LIN {X 0,Y 259.453,Z 689.028,A -85,B 0,C 180,E1 -16715.299,E2 -16715.299} C_VEL
LIN {X 0,Y 272.346,Z 664.838,A -85,B 0,C 180,E1 -16716.608,E2 -16716.608} C_VEL
LIN {X 0,Y 275.458,Z 659.109,A -85,B 0,C 180,E1 -16716.892,E2 -16716.892} C_VEL
LIN {X 0,Y 274.877,Z 634.76,A -85,B 0,C 180,E1 -16720.781,E2 -16720.781} C_VEL
LIN {X 0,Y 277.063,Z 609.313,A -85,B 0,C 180,E1 -16724.48,E2 -16724.48} C_VEL
LIN {X 0,Y 280.601,Z 587.916,A -85,B 0,C 180,E1 -16727.342,E2 -16727.342} C_VEL
LIN {X 0,Y 272.817,Z 572.023,A -85,B 0,C 180,E1 -16732.207,E2 -16732.207} C_VEL
LIN {X 0,Y 265.765,Z 558.11,A -85,B 0,C 180,E1 -16736.981,E2 -16736.981} C_VEL
LIN {X 0,Y 259.589,Z 546.11,A -85,B 0,C 180,E1 -16741.546,E2 -16741.546} C_VEL
LIN {X 0,Y 252.838,Z 533.27,A -85,B 0,C 180,E1 -16746.983,E2 -16746.983} C_VEL
LIN {X 0,Y 246.707,Z 521.951,A -85,B 0,C 180,E1 -16752.404,E2 -16752.404} C_VEL
LIN {X 0,Y 244.594,Z 517.879,A -85,B 0,C 180,E1 -16754.553,E2 -16754.553} C_VEL
LIN {X 0,Y 250.997,Z 514.698,A -85,B 0,C 180,E1 -16759.308,E2 -16759.308} C_VEL
LIN {X 0,Y 255.933,Z 513.422,A -85,B 0,C 180,E1 -16762.33,E2 -16762.33} C_VEL
LIN {X 0,Y 259.283,Z 523.373,A -85,B 0,C 180,E1 -16766.08,E2 -16766.08} C_VEL
LIN {X 0,Y 261.952,Z 531.547,A -85,B 0,C 180,E1 -16768.56,E2 -16768.56} C_VEL
LIN {X 0,Y 265.003,Z 538.596,A -85,B 0,C 180,E1 -16770.186,E2 -16770.186} C_VEL
LIN {X 0,Y 250.876,Z 717.726,A -85,B 0,C 180,E1 -16774.443,E2 -16774.443} C_VEL
LIN {X 0,Y 249.12,Z 743.516,A -85,B 0,C 180,E1 -16775.324,E2 -16775.324} C_VEL
LIN {X 0,Y 246.678,Z 762.04,A -85,B 0,C 180,E1 -16776.293,E2 -16776.293} C_VEL
LIN {X 0,Y 243.283,Z 779.25,A -85,B 0,C 180,E1 -16777.515,E2 -16777.515} C_VEL
LIN {X 0,Y 238.857,Z 796.037,A -85,B 0,C 180,E1 -16779.059,E2 -16779.059} C_VEL
LIN {X 0,Y 233.621,Z 812.02,A -85,B 0,C 180,E1 -16780.941,E2 -16780.941} C_VEL
LIN {X 0,Y 227.692,Z 827.174,A -85,B 0,C 180,E1 -16783.202,E2 -16783.202} C_VEL
LIN {X 0,Y 221.171,Z 841.428,A -85,B 0,C 180,E1 -16785.878,E2 -16785.878} C_VEL
LIN {X 0,Y 214.515,Z 854.248,A -85,B 0,C 180,E1 -16788.914,E2 -16788.914} C_VEL
LIN {X 0,Y 207.446,Z 866.472,A -85,B 0,C 180,E1 -16792.606,E2 -16792.606} C_VEL
LIN {X 0,Y 200.467,Z 877.488,A -85,B 0,C 180,E1 -16796.923,E2 -16796.923} C_VEL
LIN {X 0,Y 194.271,Z 886.647,A -85,B 0,C 180,E1 -16801.655,E2 -16801.655} C_VEL
LIN {X 0,Y 189.179,Z 893.877,A -85,B 0,C 180,E1 -16806.648,E2 -16806.648} C_VEL
LIN {X 0,Y 185.088,Z 899.588,A -85,B 0,C 180,E1 -16812.067,E2 -16812.067} C_VEL
LIN {X 0,Y 182.155,Z 903.783,A -85,B 0,C 180,E1 -16817.962,E2 -16817.962} C_VEL
LIN {X 0,Y 180.522,Z 906.241,A -85,B 0,C 180,E1 -16823.96,E2 -16823.96} C_VEL
LIN {X 0,Y 180.001,Z 907.066,A -85,B 0,C 180,E1 -16830.001,E2 -16830.001} C_VEL
LIN {X 0,Y 180.511,Z 906.288,A -85,B 0,C 180,E1 -16836.042,E2 -16836.042} C_VEL
LIN {X 0,Y 182.13,Z 903.873,A -85,B 0,C 180,E1 -16842.042,E2 -16842.042} C_VEL
LIN {X 0,Y 185.046,Z 899.716,A -85,B 0,C 180,E1 -16847.939,E2 -16847.939} C_VEL
LIN {X 0,Y 189.122,Z 894.048,A -85,B 0,C 180,E1 -16853.361,E2 -16853.361} C_VEL
LIN {X 0,Y 194.121,Z 886.989,A -85,B 0,C 180,E1 -16858.286,E2 -16858.286} C_VEL
LIN {X 0,Y 200.221,Z 878.015,A -85,B 0,C 180,E1 -16862.979,E2 -16862.979} C_VEL
LIN {X 0,Y 206.911,Z 867.529,A -85,B 0,C 180,E1 -16867.161,E2 -16867.161} C_VEL
LIN {X 0,Y 213.926,Z 855.521,A -85,B 0,C 180,E1 -16870.871,E2 -16870.871} C_VEL
LIN {X 0,Y 221.067,Z 841.893,A -85,B 0,C 180,E1 -16874.15,E2 -16874.15} C_VEL
LIN {X 0,Y 227.589,Z 827.727,A -85,B 0,C 180,E1 -16876.827,E2 -16876.827} C_VEL
LIN {X 0,Y 233.404,Z 813.001,A -85,B 0,C 180,E1 -16879.047,E2 -16879.047} C_VEL
LIN {X 0,Y 236.682,Z 803.474,A -85,B 0,C 180,E1 -16880.252,E2 -16880.252} C_VEL
LIN {X 0,Y 233.357,Z 806.151,A -85,B 0,C 180,E1 -16880.786,E2 -16880.786} C_VEL
LIN {X 0,Y 228.962,Z 810.608,A -85,B 0,C 180,E1 -16881.294,E2 -16881.294} C_VEL
LIN {X 0,Y 219.978,Z 819.575,A -85,B 0,C 180,E1 -16882.275,E2 -16882.275} C_VEL
LIN {X 0,Y 210.065,Z 829.053,A -85,B 0,C 180,E1 -16883.348,E2 -16883.348} C_VEL
LIN {X 0,Y 204.628,Z 833.297,A -85,B 0,C 180,E1 -16884.258,E2 -16884.258} C_VEL
LIN {X 0,Y 199.638,Z 836.307,A -85,B 0,C 180,E1 -16885.531,E2 -16885.531} C_VEL
LIN {X 0,Y 197.045,Z 837.699,A -85,B 0,C 180,E1 -16886.325,E2 -16886.325} C_VEL
LIN {X 0,Y 192.369,Z 840.67,A -85,B 0,C 180,E1 -16887.631,E2 -16887.631} C_VEL
LIN {X 0,Y 189.154,Z 842.143,A -85,B 0,C 180,E1 -16888.908,E2 -16888.908} C_VEL
LIN {X 0,Y 185.107,Z 844.669,A -85,B 0,C 180,E1 -16890.201,E2 -16890.201} C_VEL
LIN {X 0,Y 182.785,Z 845.372,A -85,B 0,C 180,E1 -16891.536,E2 -16891.536} C_VEL
LIN {X 0,Y 179.182,Z 860.953,A -85,B 0,C 180,E1 -16895.61,E2 -16895.61} C_VEL
LIN {X 0,Y 176.145,Z 874.608,A -85,B 0,C 180,E1 -16900.087,E2 -16900.087} C_VEL
LIN {X 0,Y 173.819,Z 886.537,A -85,B 0,C 180,E1 -16904.997,E2 -16904.997} C_VEL
LIN {X 0,Y 172.437,Z 896.396,A -85,B 0,C 180,E1 -16909.981,E2 -16909.981} C_VEL
LIN {X 0,Y 171.971,Z 905.792,A -85,B 0,C 180,E1 -16915.998,E2 -16915.998} C_VEL
LIN {X 0,Y 172.771,Z 912.99,A -85,B 0,C 180,E1 -16921.989,E2 -16921.989} C_VEL
LIN {X 0,Y 174.945,Z 918.343,A -85,B 0,C 180,E1 -16927.883,E2 -16927.883} C_VEL
LIN {X 0,Y 178.913,Z 922.183,A -85,B 0,C 180,E1 -16933.904,E2 -16933.904} C_VEL
LIN {X 0,Y 185.401,Z 924.385,A -85,B 0,C 180,E1 -16940.19,E2 -16940.19} C_VEL
LIN {X 0,Y 194.533,Z 924.651,A -85,B 0,C 180,E1 -16946.232,E2 -16946.232} C_VEL
LIN {X 0,Y 205.919,Z 923.034,A -85,B 0,C 180,E1 -16951.627,E2 -16951.627} C_VEL
LIN {X 0,Y 216.667,Z 920.548,A -85,B 0,C 180,E1 -16955.552,E2 -16955.552} C_VEL
LIN {X 0,Y 197.139,Z 933.33,A -85,B 0,C 180,E1 -16962.813,E2 -16962.813} C_VEL
LIN {X 0,Y 182.526,Z 944.843,A -85,B 0,C 180,E1 -16971.755,E2 -16971.755} C_VEL
LIN {X 0,Y 174.003,Z 953.57,A -85,B 0,C 180,E1 -16981.138,E2 -16981.138} C_VEL
LIN {X 0,Y 170.524,Z 959.101,A -85,B 0,C 180,E1 -16989.401,E2 -16989.401} C_VEL
LIN {X 0,Y 169.853,Z 962.452,A -85,B 0,C 180,E1 -16997.073,E2 -16997.073} C_VEL
LIN {X 0,Y 170.554,Z 963.775,A -85,B 0,C 180,E1 -17003.266,E2 -17003.266} C_VEL
LIN {X 0,Y 171.282,Z 963.757,A -85,B 0,C 180,E1 -17007.992,E2 -17007.992} C_VEL
LIN {X 0,Y 171.409,Z 963.117,A -85,B 0,C 180,E1 -17012.005,E2 -17012.005} C_VEL
LIN {X 0,Y 170.864,Z 961.986,A -85,B 0,C 180,E1 -17016.72,E2 -17016.72} C_VEL
LIN {X 0,Y 170.36,Z 959.287,A -85,B 0,C 180,E1 -17022.197,E2 -17022.197} C_VEL
LIN {X 0,Y 170.676,Z 954.511,A -85,B 0,C 180,E1 -17028.441,E2 -17028.441} C_VEL
LIN {X 0,Y 172.391,Z 947.879,A -85,B 0,C 180,E1 -17034.682,E2 -17034.682} C_VEL
LIN {X 0,Y 175.677,Z 939.255,A -85,B 0,C 180,E1 -17040.812,E2 -17040.812} C_VEL
LIN {X 0,Y 180.461,Z 928.724,A -85,B 0,C 180,E1 -17046.547,E2 -17046.547} C_VEL
LIN {X 0,Y 186.002,Z 917.363,A -85,B 0,C 180,E1 -17051.39,E2 -17051.39} C_VEL
LIN {X 0,Y 192.45,Z 904.191,A -85,B 0,C 180,E1 -17055.804,E2 -17055.804} C_VEL
LIN {X 0,Y 199.08,Z 890.04,A -85,B 0,C 180,E1 -17059.542,E2 -17059.542} C_VEL
LIN {X 0,Y 205.943,Z 874.399,A -85,B 0,C 180,E1 -17062.77,E2 -17062.77} C_VEL
LIN {X 0,Y 212.393,Z 857.778,A -85,B 0,C 180,E1 -17065.469,E2 -17065.469} C_VEL
LIN {X 0,Y 218.312,Z 840.21,A -85,B 0,C 180,E1 -17067.671,E2 -17067.671} C_VEL
LIN {X 0,Y 223.405,Z 822.003,A -85,B 0,C 180,E1 -17069.407,E2 -17069.407} C_VEL
LIN {X 0,Y 227.55,Z 802.864,A -85,B 0,C 180,E1 -17070.769,E2 -17070.769} C_VEL
LIN {X 0,Y 229.923,Z 789.656,A -85,B 0,C 180,E1 -17071.452,E2 -17071.452} C_VEL
LIN {X 0,Y 236.996,Z 765.246,A -85,B 0,C 180,E1 -17073.296,E2 -17073.296} C_VEL
LIN {X 0,Y 242.744,Z 741.126,A -85,B 0,C 180,E1 -17074.703,E2 -17074.703} C_VEL
LIN {X 0,Y 247.12,Z 718.034,A -85,B 0,C 180,E1 -17075.712,E2 -17075.712} C_VEL
LIN {X 0,Y 253.248,Z 689.254,A -85,B 0,C 180,E1 -17076.466,E2 -17076.466} C_VEL
LIN {X 0,Y 264.372,Z 668.041,A -85,B 0,C 180,E1 -17077.622,E2 -17077.622} C_VEL
LIN {X 0,Y 268.86,Z 660.006,A -85,B 0,C 180,E1 -17078.018,E2 -17078.018} C_VEL
LIN {X 0,Y 268.679,Z 635.94,A -85,B 0,C 180,E1 -17081.897,E2 -17081.897} C_VEL
LIN {X 0,Y 271.158,Z 610.752,A -85,B 0,C 180,E1 -17085.588,E2 -17085.588} C_VEL
LIN {X 0,Y 274.357,Z 591.962,A -85,B 0,C 180,E1 -17088.118,E2 -17088.118} C_VEL
LIN {X 0,Y 266.622,Z 576.034,A -85,B 0,C 180,E1 -17093.108,E2 -17093.108} C_VEL
LIN {X 0,Y 259.595,Z 562.101,A -85,B 0,C 180,E1 -17098.014,E2 -17098.014} C_VEL
LIN {X 0,Y 253.349,Z 550.039,A -85,B 0,C 180,E1 -17102.715,E2 -17102.715} C_VEL
LIN {X 0,Y 247.666,Z 539.087,A -85,B 0,C 180,E1 -17107.423,E2 -17107.423} C_VEL
LIN {X 0,Y 241.858,Z 528.228,A -85,B 0,C 180,E1 -17112.675,E2 -17112.675} C_VEL
LIN {X 0,Y 241.056,Z 526.523,A -85,B 0,C 180,E1 -17113.554,E2 -17113.554} C_VEL
LIN {X 0,Y 248.454,Z 522.485,A -85,B 0,C 180,E1 -17119.269,E2 -17119.269} C_VEL
LIN {X 0,Y 253,Z 521.148,A -85,B 0,C 180,E1 -17122.113,E2 -17122.113} C_VEL
LIN {X 0,Y 256.011,Z 530.778,A -85,B 0,C 180,E1 -17125.691,E2 -17125.691} C_VEL
LIN {X 0,Y 260.464,Z 541.054,A -85,B 0,C 180,E1 -17128.488,E2 -17128.488} C_VEL
LIN {X 0,Y 260.862,Z 542.461,A -85,B 0,C 180,E1 -17128.737,E2 -17128.737} C_VEL
LIN {X 0,Y 246.52,Z 718.162,A -85,B 0,C 180,E1 -17132.9,E2 -17132.9} C_VEL
LIN {X 0,Y 244.642,Z 744.592,A -85,B 0,C 180,E1 -17133.805,E2 -17133.805} C_VEL
LIN {X 0,Y 242.093,Z 763.197,A -85,B 0,C 180,E1 -17134.779,E2 -17134.779} C_VEL
LIN {X 0,Y 238.551,Z 780.49,A -85,B 0,C 180,E1 -17136.009,E2 -17136.009} C_VEL
LIN {X 0,Y 233.958,Z 797.284,A -85,B 0,C 180,E1 -17137.556,E2 -17137.556} C_VEL
LIN {X 0,Y 228.521,Z 813.273,A -85,B 0,C 180,E1 -17139.445,E2 -17139.445} C_VEL
LIN {X 0,Y 222.327,Z 828.494,A -85,B 0,C 180,E1 -17141.729,E2 -17141.729} C_VEL
LIN {X 0,Y 215.565,Z 842.687,A -85,B 0,C 180,E1 -17144.415,E2 -17144.415} C_VEL
LIN {X 0,Y 208.617,Z 855.51,A -85,B 0,C 180,E1 -17147.486,E2 -17147.486} C_VEL
LIN {X 0,Y 201.214,Z 867.737,A -85,B 0,C 180,E1 -17151.237,E2 -17151.237} C_VEL
LIN {X 0,Y 194.057,Z 878.495,A -85,B 0,C 180,E1 -17155.527,E2 -17155.527} C_VEL
LIN {X 0,Y 187.489,Z 887.699,A -85,B 0,C 180,E1 -17160.375,E2 -17160.375} C_VEL
LIN {X 0,Y 181.931,Z 895.144,A -85,B 0,C 180,E1 -17165.659,E2 -17165.659} C_VEL
LIN {X 0,Y 177.568,Z 900.855,A -85,B 0,C 180,E1 -17171.28,E2 -17171.28} C_VEL
LIN {X 0,Y 174.421,Z 905.049,A -85,B 0,C 180,E1 -17177.419,E2 -17177.419} C_VEL
LIN {X 0,Y 172.664,Z 907.505,A -85,B 0,C 180,E1 -17183.684,E2 -17183.684} C_VEL
LIN {X 0,Y 172.102,Z 908.329,A -85,B 0,C 180,E1 -17190.001,E2 -17190.001} C_VEL
LIN {X 0,Y 172.652,Z 907.552,A -85,B 0,C 180,E1 -17196.318,E2 -17196.318} C_VEL
LIN {X 0,Y 174.396,Z 905.138,A -85,B 0,C 180,E1 -17202.585,E2 -17202.585} C_VEL
LIN {X 0,Y 177.525,Z 900.981,A -85,B 0,C 180,E1 -17208.727,E2 -17208.727} C_VEL
LIN {X 0,Y 181.873,Z 895.313,A -85,B 0,C 180,E1 -17214.352,E2 -17214.352} C_VEL
LIN {X 0,Y 187.249,Z 888.153,A -85,B 0,C 180,E1 -17219.496,E2 -17219.496} C_VEL
LIN {X 0,Y 193.745,Z 879.097,A -85,B 0,C 180,E1 -17224.338,E2 -17224.338} C_VEL
LIN {X 0,Y 200.658,Z 868.788,A -85,B 0,C 180,E1 -17228.527,E2 -17228.527} C_VEL
LIN {X 0,Y 208.006,Z 856.777,A -85,B 0,C 180,E1 -17232.297,E2 -17232.297} C_VEL
LIN {X 0,Y 215.463,Z 843.146,A -85,B 0,C 180,E1 -17235.615,E2 -17235.615} C_VEL
LIN {X 0,Y 222.255,Z 828.975,A -85,B 0,C 180,E1 -17238.314,E2 -17238.314} C_VEL
LIN {X 0,Y 226.815,Z 817.853,A -85,B 0,C 180,E1 -17240.09,E2 -17240.09} C_VEL
LIN {X 0,Y 218.447,Z 823.857,A -85,B 0,C 180,E1 -17241.501,E2 -17241.501} C_VEL
LIN {X 0,Y 212.24,Z 828.459,A -85,B 0,C 180,E1 -17242.575,E2 -17242.575} C_VEL
LIN {X 0,Y 206.764,Z 831.775,A -85,B 0,C 180,E1 -17243.845,E2 -17243.845} C_VEL
LIN {X 0,Y 204.628,Z 833.297,A -85,B 0,C 180,E1 -17244.258,E2 -17244.258} C_VEL
LIN {X 0,Y 200.192,Z 836.978,A -85,B 0,C 180,E1 -17244.923,E2 -17244.923} C_VEL
LIN {X 0,Y 192.47,Z 844.021,A -85,B 0,C 180,E1 -17245.723,E2 -17245.723} C_VEL
LIN {X 0,Y 188.818,Z 846.61,A -85,B 0,C 180,E1 -17246.477,E2 -17246.477} C_VEL
LIN {X 0,Y 187.437,Z 847.296,A -85,B 0,C 180,E1 -17246.947,E2 -17246.947} C_VEL
LIN {X 0,Y 181.692,Z 850.464,A -85,B 0,C 180,E1 -17248.849,E2 -17248.849} C_VEL
LIN {X 0,Y 178.865,Z 851.626,A -85,B 0,C 180,E1 -17250.163,E2 -17250.163} C_VEL
LIN {X 0,Y 175.512,Z 853.568,A -85,B 0,C 180,E1 -17251.409,E2 -17251.409} C_VEL
LIN {X 0,Y 173.124,Z 854.331,A -85,B 0,C 180,E1 -17252.938,E2 -17252.938} C_VEL
LIN {X 0,Y 169.838,Z 868.069,A -85,B 0,C 180,E1 -17257.135,E2 -17257.135} C_VEL
LIN {X 0,Y 166.922,Z 881.484,A -85,B 0,C 180,E1 -17262.211,E2 -17262.211} C_VEL
LIN {X 0,Y 165.006,Z 892.41,A -85,B 0,C 180,E1 -17267.399,E2 -17267.399} C_VEL
LIN {X 0,Y 164.05,Z 901.947,A -85,B 0,C 180,E1 -17272.997,E2 -17272.997} C_VEL
LIN {X 0,Y 164.216,Z 910.039,A -85,B 0,C 180,E1 -17278.952,E2 -17278.952} C_VEL
LIN {X 0,Y 165.738,Z 916.608,A -85,B 0,C 180,E1 -17285.191,E2 -17285.191} C_VEL
LIN {X 0,Y 168.818,Z 921.459,A -85,B 0,C 180,E1 -17291.27,E2 -17291.27} C_VEL
LIN {X 0,Y 174.451,Z 925.045,A -85,B 0,C 180,E1 -17297.928,E2 -17297.928} C_VEL
LIN {X 0,Y 183.009,Z 926.741,A -85,B 0,C 180,E1 -17304.532,E2 -17304.532} C_VEL
LIN {X 0,Y 193.865,Z 926.488,A -85,B 0,C 180,E1 -17310.359,E2 -17310.359} C_VEL
LIN {X 0,Y 206.674,Z 924.609,A -85,B 0,C 180,E1 -17315.393,E2 -17315.393} C_VEL
LIN {X 0,Y 187.182,Z 936.381,A -85,B 0,C 180,E1 -17323.135,E2 -17323.135} C_VEL
LIN {X 0,Y 172.614,Z 947.012,A -85,B 0,C 180,E1 -17332.956,E2 -17332.956} C_VEL
LIN {X 0,Y 165.051,Z 954.434,A -85,B 0,C 180,E1 -17342.586,E2 -17342.586} C_VEL
LIN {X 0,Y 162.169,Z 959.206,A -85,B 0,C 180,E1 -17351.709,E2 -17351.709} C_VEL
LIN {X 0,Y 162.157,Z 961.558,A -85,B 0,C 180,E1 -17359.339,E2 -17359.339} C_VEL
LIN {X 0,Y 163.119,Z 962.109,A -85,B 0,C 180,E1 -17365.429,E2 -17365.429} C_VEL
LIN {X 0,Y 163.577,Z 962.001,A -85,B 0,C 180,E1 -17369.649,E2 -17369.649} C_VEL
LIN {X 0,Y 163.283,Z 961.502,A -85,B 0,C 180,E1 -17374.213,E2 -17374.213} C_VEL
LIN {X 0,Y 162.602,Z 959.699,A -85,B 0,C 180,E1 -17379.556,E2 -17379.556} C_VEL
LIN {X 0,Y 162.429,Z 956.059,A -85,B 0,C 180,E1 -17385.714,E2 -17385.714} C_VEL
LIN {X 0,Y 163.527,Z 950.451,A -85,B 0,C 180,E1 -17392.276,E2 -17392.276} C_VEL
LIN {X 0,Y 166.231,Z 942.942,A -85,B 0,C 180,E1 -17398.762,E2 -17398.762} C_VEL
LIN {X 0,Y 170.682,Z 933.375,A -85,B 0,C 180,E1 -17405.034,E2 -17405.034} C_VEL
LIN {X 0,Y 176.497,Z 922.135,A -85,B 0,C 180,E1 -17410.652,E2 -17410.652} C_VEL
LIN {X 0,Y 182.851,Z 910.179,A -85,B 0,C 180,E1 -17415.304,E2 -17415.304} C_VEL
LIN {X 0,Y 189.941,Z 896.371,A -85,B 0,C 180,E1 -17419.51,E2 -17419.51} C_VEL
LIN {X 0,Y 197.142,Z 881.561,A -85,B 0,C 180,E1 -17423.015,E2 -17423.015} C_VEL
LIN {X 0,Y 203.983,Z 865.913,A -85,B 0,C 180,E1 -17425.932,E2 -17425.932} C_VEL
LIN {X 0,Y 210.594,Z 849.03,A -85,B 0,C 180,E1 -17428.339,E2 -17428.339} C_VEL
LIN {X 0,Y 216.033,Z 832.473,A -85,B 0,C 180,E1 -17430.203,E2 -17430.203} C_VEL
LIN {X 0,Y 220.972,Z 814.096,A -85,B 0,C 180,E1 -17431.77,E2 -17431.77} C_VEL
LIN {X 0,Y 224.854,Z 795.017,A -85,B 0,C 180,E1 -17432.946,E2 -17432.946} C_VEL
LIN {X 0,Y 227.381,Z 776.929,A -85,B 0,C 180,E1 -17433.691,E2 -17433.691} C_VEL
LIN {X 0,Y 227.896,Z 774.037,A -85,B 0,C 180,E1 -17433.793,E2 -17433.793} C_VEL
LIN {X 0,Y 234.313,Z 750.257,A -85,B 0,C 180,E1 -17435.354,E2 -17435.354} C_VEL
LIN {X 0,Y 239.535,Z 725.305,A -85,B 0,C 180,E1 -17436.638,E2 -17436.638} C_VEL
LIN {X 0,Y 245.17,Z 698.026,A -85,B 0,C 180,E1 -17437.493,E2 -17437.493} C_VEL
LIN {X 0,Y 247.908,Z 687.006,A -85,B 0,C 180,E1 -17437.76,E2 -17437.76} C_VEL
LIN {X 0,Y 260.742,Z 663.573,A -85,B 0,C 180,E1 -17439.024,E2 -17439.024} C_VEL
LIN {X 0,Y 262.255,Z 660.786,A -85,B 0,C 180,E1 -17439.17,E2 -17439.17} C_VEL
LIN {X 0,Y 262.516,Z 636.111,A -85,B 0,C 180,E1 -17443.175,E2 -17443.175} C_VEL
LIN {X 0,Y 265.491,Z 610.547,A -85,B 0,C 180,E1 -17446.941,E2 -17446.941} C_VEL
LIN {X 0,Y 268.15,Z 596.033,A -85,B 0,C 180,E1 -17448.929,E2 -17448.929} C_VEL
LIN {X 0,Y 260.353,Z 579.937,A -85,B 0,C 180,E1 -17454.074,E2 -17454.074} C_VEL
LIN {X 0,Y 253.343,Z 565.941,A -85,B 0,C 180,E1 -17459.096,E2 -17459.096} C_VEL
LIN {X 0,Y 246.867,Z 553.291,A -85,B 0,C 180,E1 -17464.181,E2 -17464.181} C_VEL
LIN {X 0,Y 240.905,Z 541.877,A -85,B 0,C 180,E1 -17469.316,E2 -17469.316} C_VEL
LIN {X 0,Y 237.575,Z 535.424,A -85,B 0,C 180,E1 -17472.519,E2 -17472.519} C_VEL
LIN {X 0,Y 244.282,Z 531.125,A -85,B 0,C 180,E1 -17478.125,E2 -17478.125} C_VEL
LIN {X 0,Y 250.092,Z 529.021,A -85,B 0,C 180,E1 -17481.906,E2 -17481.906} C_VEL
LIN {X 0,Y 252.142,Z 535.031,A -85,B 0,C 180,E1 -17484.17,E2 -17484.17} C_VEL
LIN {X 0,Y 256.923,Z 545.991,A -85,B 0,C 180,E1 -17487.236,E2 -17487.236} C_VEL
LIN {X 0,Y 242.344,Z 718.695,A -85,B 0,C 180,E1 -17491.305,E2 -17491.305} C_VEL
LIN {X 0,Y 240.325,Z 745.803,A -85,B 0,C 180,E1 -17492.236,E2 -17492.236} C_VEL
LIN {X 0,Y 237.67,Z 764.427,A -85,B 0,C 180,E1 -17493.213,E2 -17493.213} C_VEL
LIN {X 0,Y 233.992,Z 781.731,A -85,B 0,C 180,E1 -17494.443,E2 -17494.443} C_VEL
LIN {X 0,Y 229.218,Z 798.562,A -85,B 0,C 180,E1 -17495.994,E2 -17495.994} C_VEL
LIN {X 0,Y 223.584,Z 814.525,A -85,B 0,C 180,E1 -17497.881,E2 -17497.881} C_VEL
LIN {X 0,Y 217.177,Z 829.686,A -85,B 0,C 180,E1 -17500.161,E2 -17500.161} C_VEL
LIN {X 0,Y 210.047,Z 844.059,A -85,B 0,C 180,E1 -17502.9,E2 -17502.9} C_VEL
LIN {X 0,Y 202.556,Z 857.262,A -85,B 0,C 180,E1 -17506.112,E2 -17506.112} C_VEL
LIN {X 0,Y 195.102,Z 869.005,A -85,B 0,C 180,E1 -17509.783,E2 -17509.783} C_VEL
LIN {X 0,Y 187.643,Z 879.675,A -85,B 0,C 180,E1 -17514.118,E2 -17514.118} C_VEL
LIN {X 0,Y 180.755,Z 888.819,A -85,B 0,C 180,E1 -17519.041,E2 -17519.041} C_VEL
LIN {X 0,Y 174.741,Z 896.412,A -85,B 0,C 180,E1 -17524.588,E2 -17524.588} C_VEL
LIN {X 0,Y 170.084,Z 902.123,A -85,B 0,C 180,E1 -17530.423,E2 -17530.423} C_VEL
LIN {X 0,Y 166.706,Z 906.315,A -85,B 0,C 180,E1 -17536.827,E2 -17536.827} C_VEL
LIN {X 0,Y 164.809,Z 908.769,A -85,B 0,C 180,E1 -17543.382,E2 -17543.382} C_VEL
LIN {X 0,Y 164.203,Z 909.592,A -85,B 0,C 180,E1 -17550.001,E2 -17550.001} C_VEL
LIN {X 0,Y 164.797,Z 908.816,A -85,B 0,C 180,E1 -17556.621,E2 -17556.621} C_VEL
LIN {X 0,Y 166.679,Z 906.403,A -85,B 0,C 180,E1 -17563.178,E2 -17563.178} C_VEL
LIN {X 0,Y 170.04,Z 902.246,A -85,B 0,C 180,E1 -17569.584,E2 -17569.584} C_VEL
LIN {X 0,Y 174.682,Z 896.578,A -85,B 0,C 180,E1 -17575.424,E2 -17575.424} C_VEL
LIN {X 0,Y 180.55,Z 889.21,A -85,B 0,C 180,E1 -17580.864,E2 -17580.864} C_VEL
LIN {X 0,Y 187.436,Z 880.111,A -85,B 0,C 180,E1 -17585.821,E2 -17585.821} C_VEL
LIN {X 0,Y 195.016,Z 869.316,A -85,B 0,C 180,E1 -17590.242,E2 -17590.242} C_VEL
LIN {X 0,Y 202.762,Z 857.151,A -85,B 0,C 180,E1 -17594.052,E2 -17594.052} C_VEL
LIN {X 0,Y 210.297,Z 843.866,A -85,B 0,C 180,E1 -17597.272,E2 -17597.272} C_VEL
LIN {X 0,Y 217.347,Z 829.617,A -85,B 0,C 180,E1 -17599.983,E2 -17599.983} C_VEL
LIN {X 0,Y 210.401,Z 834.274,A -85,B 0,C 180,E1 -17601.149,E2 -17601.149} C_VEL
LIN {X 0,Y 205.562,Z 837.102,A -85,B 0,C 180,E1 -17602.202,E2 -17602.202} C_VEL
LIN {X 0,Y 199.647,Z 840.78,A -85,B 0,C 180,E1 -17603.417,E2 -17603.417} C_VEL
LIN {X 0,Y 195.256,Z 843.018,A -85,B 0,C 180,E1 -17604.644,E2 -17604.644} C_VEL
LIN {X 0,Y 189.862,Z 846.195,A -85,B 0,C 180,E1 -17606.066,E2 -17606.066} C_VEL
LIN {X 0,Y 187.437,Z 847.296,A -85,B 0,C 180,E1 -17606.947,E2 -17606.947} C_VEL
LIN {X 0,Y 183.898,Z 849.2,A -85,B 0,C 180,E1 -17608.14,E2 -17608.14} C_VEL
LIN {X 0,Y 177.553,Z 853.705,A -85,B 0,C 180,E1 -17609.613,E2 -17609.613} C_VEL
LIN {X 0,Y 169.723,Z 859.465,A -85,B 0,C 180,E1 -17611.455,E2 -17611.455} C_VEL
LIN {X 0,Y 165.662,Z 861.906,A -85,B 0,C 180,E1 -17612.992,E2 -17612.992} C_VEL
LIN {X 0,Y 164.101,Z 862.564,A -85,B 0,C 180,E1 -17613.953,E2 -17613.953} C_VEL
LIN {X 0,Y 163.408,Z 862.746,A -85,B 0,C 180,E1 -17614.638,E2 -17614.638} C_VEL
LIN {X 0,Y 160.168,Z 876.453,A -85,B 0,C 180,E1 -17619.537,E2 -17619.537} C_VEL
LIN {X 0,Y 157.725,Z 888.489,A -85,B 0,C 180,E1 -17624.934,E2 -17624.934} C_VEL
LIN {X 0,Y 156.29,Z 899.073,A -85,B 0,C 180,E1 -17630.796,E2 -17630.796} C_VEL
LIN {X 0,Y 156.1,Z 908.943,A -85,B 0,C 180,E1 -17637.759,E2 -17637.759} C_VEL
LIN {X 0,Y 157.464,Z 916.323,A -85,B 0,C 180,E1 -17644.491,E2 -17644.491} C_VEL
LIN {X 0,Y 160.38,Z 921.667,A -85,B 0,C 180,E1 -17650.778,E2 -17650.778} C_VEL
LIN {X 0,Y 165.731,Z 925.872,A -85,B 0,C 180,E1 -17657.556,E2 -17657.556} C_VEL
LIN {X 0,Y 174.162,Z 928.39,A -85,B 0,C 180,E1 -17664.414,E2 -17664.414} C_VEL
LIN {X 0,Y 185.623,Z 928.956,A -85,B 0,C 180,E1 -17670.777,E2 -17670.777} C_VEL
LIN {X 0,Y 196.53,Z 928.096,A -85,B 0,C 180,E1 -17675.257,E2 -17675.257} C_VEL
LIN {X 0,Y 177.223,Z 938.84,A -85,B 0,C 180,E1 -17683.494,E2 -17683.494} C_VEL
LIN {X 0,Y 163.47,Z 948.143,A -85,B 0,C 180,E1 -17693.607,E2 -17693.607} C_VEL
LIN {X 0,Y 156.384,Z 954.604,A -85,B 0,C 180,E1 -17703.821,E2 -17703.821} C_VEL
LIN {X 0,Y 154.141,Z 958.434,A -85,B 0,C 180,E1 -17713.027,E2 -17713.027} C_VEL
LIN {X 0,Y 154.495,Z 960.084,A -85,B 0,C 180,E1 -17720.688,E2 -17720.688} C_VEL
LIN {X 0,Y 155.463,Z 960.476,A -85,B 0,C 180,E1 -17726.681,E2 -17726.681} C_VEL
LIN {X 0,Y 155.66,Z 960.677,A -85,B 0,C 180,E1 -17731.103,E2 -17731.103} C_VEL
LIN {X 0,Y 155.167,Z 959.954,A -85,B 0,C 180,E1 -17735.546,E2 -17735.546} C_VEL
LIN {X 0,Y 154.498,Z 957.658,A -85,B 0,C 180,E1 -17741.572,E2 -17741.572} C_VEL
LIN {X 0,Y 154.713,Z 953.352,A -85,B 0,C 180,E1 -17748.461,E2 -17748.461} C_VEL
LIN {X 0,Y 156.517,Z 947.21,A -85,B 0,C 180,E1 -17755.34,E2 -17755.34} C_VEL
LIN {X 0,Y 160.101,Z 939.123,A -85,B 0,C 180,E1 -17762.061,E2 -17762.061} C_VEL
LIN {X 0,Y 165.54,Z 928.908,A -85,B 0,C 180,E1 -17768.47,E2 -17768.47} C_VEL
LIN {X 0,Y 171.948,Z 917.648,A -85,B 0,C 180,E1 -17773.86,E2 -17773.86} C_VEL
LIN {X 0,Y 178.994,Z 905.236,A -85,B 0,C 180,E1 -17778.461,E2 -17778.461} C_VEL
LIN {X 0,Y 186.559,Z 891.272,A -85,B 0,C 180,E1 -17782.485,E2 -17782.485} C_VEL
LIN {X 0,Y 194.367,Z 875.796,A -85,B 0,C 180,E1 -17785.914,E2 -17785.914} C_VEL
LIN {X 0,Y 201.407,Z 860.042,A -85,B 0,C 180,E1 -17788.634,E2 -17788.634} C_VEL
LIN {X 0,Y 208.185,Z 842.685,A -85,B 0,C 180,E1 -17790.937,E2 -17790.937} C_VEL
LIN {X 0,Y 214.141,Z 824.348,A -85,B 0,C 180,E1 -17792.77,E2 -17792.77} C_VEL
LIN {X 0,Y 218.854,Z 805.948,A -85,B 0,C 180,E1 -17794.14,E2 -17794.14} C_VEL
LIN {X 0,Y 222.304,Z 787.72,A -85,B 0,C 180,E1 -17795.11,E2 -17795.11} C_VEL
LIN {X 0,Y 224.657,Z 767.989,A -85,B 0,C 180,E1 -17795.805,E2 -17795.805} C_VEL
LIN {X 0,Y 225.699,Z 758.634,A -85,B 0,C 180,E1 -17796.02,E2 -17796.02} C_VEL
LIN {X 0,Y 231.453,Z 734.566,A -85,B 0,C 180,E1 -17797.418,E2 -17797.418} C_VEL
LIN {X 0,Y 236.026,Z 712.171,A -85,B 0,C 180,E1 -17798.352,E2 -17798.352} C_VEL
LIN {X 0,Y 242.002,Z 686.439,A -85,B 0,C 180,E1 -17799.025,E2 -17799.025} C_VEL
LIN {X 0,Y 254.914,Z 663.06,A -85,B 0,C 180,E1 -17800.28,E2 -17800.28} C_VEL
LIN {X 0,Y 255.729,Z 661.611,A -85,B 0,C 180,E1 -17800.352,E2 -17800.352} C_VEL
LIN {X 0,Y 256.407,Z 636.891,A -85,B 0,C 180,E1 -17804.401,E2 -17804.401} C_VEL
LIN {X 0,Y 259.943,Z 610.207,A -85,B 0,C 180,E1 -17808.35,E2 -17808.35} C_VEL
LIN {X 0,Y 261.844,Z 599.967,A -85,B 0,C 180,E1 -17809.773,E2 -17809.773} C_VEL
LIN {X 0,Y 254.42,Z 584.512,A -85,B 0,C 180,E1 -17814.815,E2 -17814.815} C_VEL
LIN {X 0,Y 247.4,Z 570.412,A -85,B 0,C 180,E1 -17820.001,E2 -17820.001} C_VEL
LIN {X 0,Y 241.493,Z 558.775,A -85,B 0,C 180,E1 -17824.751,E2 -17824.751} C_VEL
LIN {X 0,Y 235.786,Z 547.733,A -85,B 0,C 180,E1 -17829.766,E2 -17829.766} C_VEL
LIN {X 0,Y 234.295,Z 544.926,A -85,B 0,C 180,E1 -17831.185,E2 -17831.185} C_VEL
LIN {X 0,Y 239.023,Z 540.706,A -85,B 0,C 180,E1 -17835.778,E2 -17835.778} C_VEL
LIN {X 0,Y 245.927,Z 537.456,A -85,B 0,C 180,E1 -17840.715,E2 -17840.715} C_VEL
LIN {X 0,Y 247.531,Z 537.011,A -85,B 0,C 180,E1 -17841.692,E2 -17841.692} C_VEL
LIN {X 0,Y 251.435,Z 545.771,A -85,B 0,C 180,E1 -17844.555,E2 -17844.555} C_VEL
LIN {X 0,Y 253.12,Z 550.021,A -85,B 0,C 180,E1 -17845.7,E2 -17845.7} C_VEL
LIN {X 0,Y 238.363,Z 719.217,A -85,B 0,C 180,E1 -17849.655,E2 -17849.655} C_VEL
LIN {X 0,Y 236.215,Z 746.855,A -85,B 0,C 180,E1 -17850.604,E2 -17850.604} C_VEL
LIN {X 0,Y 233.451,Z 765.552,A -85,B 0,C 180,E1 -17851.581,E2 -17851.581} C_VEL
LIN {X 0,Y 229.613,Z 782.971,A -85,B 0,C 180,E1 -17852.816,E2 -17852.816} C_VEL
LIN {X 0,Y 224.675,Z 799.779,A -85,B 0,C 180,E1 -17854.36,E2 -17854.36} C_VEL
LIN {X 0,Y 218.821,Z 815.778,A -85,B 0,C 180,E1 -17856.248,E2 -17856.248} C_VEL
LIN {X 0,Y 212.166,Z 830.942,A -85,B 0,C 180,E1 -17858.53,E2 -17858.53} C_VEL
LIN {X 0,Y 204.81,Z 845.205,A -85,B 0,C 180,E1 -17861.254,E2 -17861.254} C_VEL
LIN {X 0,Y 197.164,Z 858.16,A -85,B 0,C 180,E1 -17864.414,E2 -17864.414} C_VEL
LIN {X 0,Y 189.129,Z 870.264,A -85,B 0,C 180,E1 -17868.233,E2 -17868.233} C_VEL
LIN {X 0,Y 181.286,Z 880.94,A -85,B 0,C 180,E1 -17872.65,E2 -17872.65} C_VEL
LIN {X 0,Y 174.008,Z 890.086,A -85,B 0,C 180,E1 -17877.699,E2 -17877.699} C_VEL
LIN {X 0,Y 167.617,Z 897.679,A -85,B 0,C 180,E1 -17883.425,E2 -17883.425} C_VEL
LIN {X 0,Y 162.641,Z 903.39,A -85,B 0,C 180,E1 -17889.488,E2 -17889.488} C_VEL
LIN {X 0,Y 159.008,Z 907.582,A -85,B 0,C 180,E1 -17896.177,E2 -17896.177} C_VEL
LIN {X 0,Y 156.96,Z 910.034,A -85,B 0,C 180,E1 -17903.049,E2 -17903.049} C_VEL
LIN {X 0,Y 156.303,Z 910.855,A -85,B 0,C 180,E1 -17910.001,E2 -17910.001} C_VEL
LIN {X 0,Y 156.947,Z 910.079,A -85,B 0,C 180,E1 -17916.953,E2 -17916.953} C_VEL
LIN {X 0,Y 158.981,Z 907.668,A -85,B 0,C 180,E1 -17923.828,E2 -17923.828} C_VEL
LIN {X 0,Y 162.597,Z 903.512,A -85,B 0,C 180,E1 -17930.52,E2 -17930.52} C_VEL
LIN {X 0,Y 167.557,Z 897.843,A -85,B 0,C 180,E1 -17936.587,E2 -17936.587} C_VEL
LIN {X 0,Y 173.548,Z 890.78,A -85,B 0,C 180,E1 -17942.009,E2 -17942.009} C_VEL
LIN {X 0,Y 180.746,Z 881.8,A -85,B 0,C 180,E1 -17947.084,E2 -17947.084} C_VEL
LIN {X 0,Y 188.528,Z 871.307,A -85,B 0,C 180,E1 -17951.526,E2 -17951.526} C_VEL
LIN {X 0,Y 196.709,Z 859.101,A -85,B 0,C 180,E1 -17955.456,E2 -17955.456} C_VEL
LIN {X 0,Y 204.713,Z 845.649,A -85,B 0,C 180,E1 -17958.78,E2 -17958.78} C_VEL
LIN {X 0,Y 207.497,Z 840.453,A -85,B 0,C 180,E1 -17959.871,E2 -17959.871} C_VEL
LIN {X 0,Y 203.44,Z 842.799,A -85,B 0,C 180,E1 -17960.653,E2 -17960.653} C_VEL
LIN {X 0,Y 196.326,Z 846.827,A -85,B 0,C 180,E1 -17962.13,E2 -17962.13} C_VEL
LIN {X 0,Y 192.592,Z 848.692,A -85,B 0,C 180,E1 -17963.084,E2 -17963.084} C_VEL
LIN {X 0,Y 186.624,Z 851.859,A -85,B 0,C 180,E1 -17964.645,E2 -17964.645} C_VEL
LIN {X 0,Y 183.173,Z 853.453,A -85,B 0,C 180,E1 -17965.789,E2 -17965.789} C_VEL
LIN {X 0,Y 178.188,Z 856.047,A -85,B 0,C 180,E1 -17967.405,E2 -17967.405} C_VEL
LIN {X 0,Y 175.107,Z 857.375,A -85,B 0,C 180,E1 -17968.693,E2 -17968.693} C_VEL
LIN {X 0,Y 170.632,Z 859.572,A -85,B 0,C 180,E1 -17970.513,E2 -17970.513} C_VEL
LIN {X 0,Y 168.842,Z 860.236,A -85,B 0,C 180,E1 -17971.528,E2 -17971.528} C_VEL
LIN {X 0,Y 165.445,Z 862.06,A -85,B 0,C 180,E1 -17973.046,E2 -17973.046} C_VEL
LIN {X 0,Y 164.101,Z 862.564,A -85,B 0,C 180,E1 -17973.953,E2 -17973.953} C_VEL
LIN {X 0,Y 163.088,Z 863.476,A -85,B 0,C 180,E1 -17974.699,E2 -17974.699} C_VEL
LIN {X 0,Y 159.212,Z 870.237,A -85,B 0,C 180,E1 -17976.933,E2 -17976.933} C_VEL
LIN {X 0,Y 152.725,Z 880.002,A -85,B 0,C 180,E1 -17980.355,E2 -17980.355} C_VEL
LIN {X 0,Y 150.501,Z 885.003,A -85,B 0,C 180,E1 -17982.71,E2 -17982.71} C_VEL
LIN {X 0,Y 148.632,Z 896.242,A -85,B 0,C 180,E1 -17988.749,E2 -17988.749} C_VEL
LIN {X 0,Y 147.989,Z 906.101,A -85,B 0,C 180,E1 -17995.348,E2 -17995.348} C_VEL
LIN {X 0,Y 148.735,Z 913.951,A -85,B 0,C 180,E1 -18001.925,E2 -18001.925} C_VEL
LIN {X 0,Y 151.52,Z 921.047,A -85,B 0,C 180,E1 -18009.494,E2 -18009.494} C_VEL
LIN {X 0,Y 156.893,Z 926.307,A -85,B 0,C 180,E1 -18017.046,E2 -18017.046} C_VEL
LIN {X 0,Y 165.266,Z 929.673,A -85,B 0,C 180,E1 -18024.292,E2 -18024.292} C_VEL
LIN {X 0,Y 176.782,Z 931.13,A -85,B 0,C 180,E1 -18030.975,E2 -18030.975} C_VEL
LIN {X 0,Y 186.384,Z 931.068,A -85,B 0,C 180,E1 -18035.125,E2 -18035.125} C_VEL
LIN {X 0,Y 167.012,Z 940.975,A -85,B 0,C 180,E1 -18044.075,E2 -18044.075} C_VEL
LIN {X 0,Y 153.719,Z 949.251,A -85,B 0,C 180,E1 -18055.082,E2 -18055.082} C_VEL
LIN {X 0,Y 147.545,Z 954.739,A -85,B 0,C 180,E1 -18066.007,E2 -18066.007} C_VEL
LIN {X 0,Y 146.207,Z 957.511,A -85,B 0,C 180,E1 -18075.342,E2 -18075.342} C_VEL
LIN {X 0,Y 147.103,Z 958.501,A -85,B 0,C 180,E1 -18083.364,E2 -18083.364} C_VEL
LIN {X 0,Y 147.694,Z 959.353,A -85,B 0,C 180,E1 -18088.059,E2 -18088.059} C_VEL
LIN {X 0,Y 147.697,Z 959.35,A -85,B 0,C 180,E1 -18091.939,E2 -18091.939} C_VEL
LIN {X 0,Y 147.02,Z 958.387,A -85,B 0,C 180,E1 -18097.03,E2 -18097.03} C_VEL
LIN {X 0,Y 146.473,Z 955.76,A -85,B 0,C 180,E1 -18103.419,E2 -18103.419} C_VEL
LIN {X 0,Y 147.109,Z 951.131,A -85,B 0,C 180,E1 -18110.696,E2 -18110.696} C_VEL
LIN {X 0,Y 149.524,Z 944.663,A -85,B 0,C 180,E1 -18117.909,E2 -18117.909} C_VEL
LIN {X 0,Y 153.592,Z 936.756,A -85,B 0,C 180,E1 -18124.495,E2 -18124.495} C_VEL
LIN {X 0,Y 159.394,Z 926.931,A -85,B 0,C 180,E1 -18130.72,E2 -18130.72} C_VEL
LIN {X 0,Y 166.358,Z 915.669,A -85,B 0,C 180,E1 -18136.155,E2 -18136.155} C_VEL
LIN {X 0,Y 174.038,Z 902.987,A -85,B 0,C 180,E1 -18140.857,E2 -18140.857} C_VEL
LIN {X 0,Y 182.168,Z 888.867,A -85,B 0,C 180,E1 -18144.865,E2 -18144.865} C_VEL
LIN {X 0,Y 190.432,Z 873.161,A -85,B 0,C 180,E1 -18148.273,E2 -18148.273} C_VEL
LIN {X 0,Y 197.91,Z 857.156,A -85,B 0,C 180,E1 -18150.927,E2 -18150.927} C_VEL
LIN {X 0,Y 204.644,Z 840.38,A -85,B 0,C 180,E1 -18153.082,E2 -18153.082} C_VEL
LIN {X 0,Y 210.53,Z 822.89,A -85,B 0,C 180,E1 -18154.786,E2 -18154.786} C_VEL
LIN {X 0,Y 215.538,Z 803.979,A -85,B 0,C 180,E1 -18156.153,E2 -18156.153} C_VEL
LIN {X 0,Y 219.219,Z 784.874,A -85,B 0,C 180,E1 -18157.119,E2 -18157.119} C_VEL
LIN {X 0,Y 221.574,Z 765.671,A -85,B 0,C 180,E1 -18157.741,E2 -18157.741} C_VEL
LIN {X 0,Y 224.181,Z 739.215,A -85,B 0,C 180,E1 -18158.421,E2 -18158.421} C_VEL
LIN {X 0,Y 229.102,Z 715.982,A -85,B 0,C 180,E1 -18159.499,E2 -18159.499} C_VEL
LIN {X 0,Y 235.842,Z 686.658,A -85,B 0,C 180,E1 -18160.293,E2 -18160.293} C_VEL
LIN {X 0,Y 244.982,Z 669.648,A -85,B 0,C 180,E1 -18161.239,E2 -18161.239} C_VEL
LIN {X 0,Y 249.263,Z 662.161,A -85,B 0,C 180,E1 -18161.617,E2 -18161.617} C_VEL
LIN {X 0,Y 250.352,Z 637.656,A -85,B 0,C 180,E1 -18165.664,E2 -18165.664} C_VEL
LIN {X 0,Y 254.347,Z 610.565,A -85,B 0,C 180,E1 -18169.697,E2 -18169.697} C_VEL
LIN {X 0,Y 255.551,Z 603.926,A -85,B 0,C 180,E1 -18170.656,E2 -18170.656} C_VEL
LIN {X 0,Y 248.443,Z 588.993,A -85,B 0,C 180,E1 -18175.615,E2 -18175.615} C_VEL
LIN {X 0,Y 241.697,Z 575.352,A -85,B 0,C 180,E1 -18180.712,E2 -18180.712} C_VEL
LIN {X 0,Y 235.502,Z 563.063,A -85,B 0,C 180,E1 -18185.849,E2 -18185.849} C_VEL
LIN {X 0,Y 231.729,Z 555.601,A -85,B 0,C 180,E1 -18189.312,E2 -18189.312} C_VEL
LIN {X 0,Y 233.503,Z 553.065,A -85,B 0,C 180,E1 -18191.486,E2 -18191.486} C_VEL
LIN {X 0,Y 237.255,Z 549.326,A -85,B 0,C 180,E1 -18195.147,E2 -18195.147} C_VEL
LIN {X 0,Y 244.665,Z 545.506,A -85,B 0,C 180,E1 -18200.577,E2 -18200.577} C_VEL
LIN {X 0,Y 246.044,Z 545.418,A -85,B 0,C 180,E1 -18201.454,E2 -18201.454} C_VEL
LIN {X 0,Y 249.52,Z 553.818,A -85,B 0,C 180,E1 -18204.11,E2 -18204.11} C_VEL
LIN {X 0,Y 234.584,Z 719.767,A -85,B 0,C 180,E1 -18207.952,E2 -18207.952} C_VEL
LIN {X 0,Y 232.284,Z 748.06,A -85,B 0,C 180,E1 -18208.922,E2 -18208.922} C_VEL
LIN {X 0,Y 229.407,Z 766.78,A -85,B 0,C 180,E1 -18209.898,E2 -18209.898} C_VEL
LIN {X 0,Y 225.427,Z 784.211,A -85,B 0,C 180,E1 -18211.127,E2 -18211.127} C_VEL
LIN {X 0,Y 220.111,Z 801.59,A -85,B 0,C 180,E1 -18212.723,E2 -18212.723} C_VEL
LIN {X 0,Y 213.91,Z 817.809,A -85,B 0,C 180,E1 -18214.649,E2 -18214.649} C_VEL
LIN {X 0,Y 206.684,Z 833.478,A -85,B 0,C 180,E1 -18217.042,E2 -18217.042} C_VEL
LIN {X 0,Y 198.604,Z 848.307,A -85,B 0,C 180,E1 -18219.955,E2 -18219.955} C_VEL
LIN {X 0,Y 190.622,Z 861.061,A -85,B 0,C 180,E1 -18223.191,E2 -18223.191} C_VEL
LIN {X 0,Y 182.224,Z 872.992,A -85,B 0,C 180,E1 -18227.127,E2 -18227.127} C_VEL
LIN {X 0,Y 174.092,Z 883.408,A -85,B 0,C 180,E1 -18231.665,E2 -18231.665} C_VEL
LIN {X 0,Y 166.54,Z 892.321,A -85,B 0,C 180,E1 -18236.885,E2 -18236.885} C_VEL
LIN {X 0,Y 159.908,Z 899.703,A -85,B 0,C 180,E1 -18242.843,E2 -18242.843} C_VEL
LIN {X 0,Y 154.515,Z 905.457,A -85,B 0,C 180,E1 -18249.549,E2 -18249.549} C_VEL
LIN {X 0,Y 150.873,Z 909.337,A -85,B 0,C 180,E1 -18256.589,E2 -18256.589} C_VEL
LIN {X 0,Y 148.9,Z 911.508,A -85,B 0,C 180,E1 -18263.833,E2 -18263.833} C_VEL
LIN {X 0,Y 148.408,Z 912.087,A -85,B 0,C 180,E1 -18270.773,E2 -18270.773} C_VEL
LIN {X 0,Y 149.178,Z 911.241,A -85,B 0,C 180,E1 -18277.705,E2 -18277.705} C_VEL
LIN {X 0,Y 151.464,Z 908.743,A -85,B 0,C 180,E1 -18284.92,E2 -18284.92} C_VEL
LIN {X 0,Y 155.453,Z 904.496,A -85,B 0,C 180,E1 -18291.905,E2 -18291.905} C_VEL
LIN {X 0,Y 160.845,Z 898.73,A -85,B 0,C 180,E1 -18298.194,E2 -18298.194} C_VEL
LIN {X 0,Y 167.71,Z 891.077,A -85,B 0,C 180,E1 -18304.086,E2 -18304.086} C_VEL
LIN {X 0,Y 175.463,Z 881.859,A -85,B 0,C 180,E1 -18309.238,E2 -18309.238} C_VEL
LIN {X 0,Y 183.76,Z 871.102,A -85,B 0,C 180,E1 -18313.712,E2 -18313.712} C_VEL
LIN {X 0,Y 191.704,Z 859.662,A -85,B 0,C 180,E1 -18317.343,E2 -18317.343} C_VEL
LIN {X 0,Y 197.507,Z 850.382,A -85,B 0,C 180,E1 -18319.739,E2 -18319.739} C_VEL
LIN {X 0,Y 189.62,Z 854.27,A -85,B 0,C 180,E1 -18321.521,E2 -18321.521} C_VEL
LIN {X 0,Y 183.337,Z 857.307,A -85,B 0,C 180,E1 -18323.136,E2 -18323.136} C_VEL
LIN {X 0,Y 179.665,Z 858.986,A -85,B 0,C 180,E1 -18324.243,E2 -18324.243} C_VEL
LIN {X 0,Y 173.961,Z 861.644,A -85,B 0,C 180,E1 -18326.115,E2 -18326.115} C_VEL
LIN {X 0,Y 171.327,Z 862.8,A -85,B 0,C 180,E1 -18327.128,E2 -18327.128} C_VEL
LIN {X 0,Y 166.2,Z 865.099,A -85,B 0,C 180,E1 -18329.244,E2 -18329.244} C_VEL
LIN {X 0,Y 164.453,Z 865.822,A -85,B 0,C 180,E1 -18330.095,E2 -18330.095} C_VEL
LIN {X 0,Y 160.295,Z 867.746,A -85,B 0,C 180,E1 -18332.106,E2 -18332.106} C_VEL
LIN {X 0,Y 158.356,Z 868.49,A -85,B 0,C 180,E1 -18333.365,E2 -18333.365} C_VEL
LIN {X 0,Y 155.096,Z 870.112,A -85,B 0,C 180,E1 -18335.225,E2 -18335.225} C_VEL
LIN {X 0,Y 153.738,Z 870.68,A -85,B 0,C 180,E1 -18336.625,E2 -18336.625} C_VEL
LIN {X 0,Y 150.707,Z 884.007,A -85,B 0,C 180,E1 -18342.23,E2 -18342.23} C_VEL
LIN {X 0,Y 150.501,Z 885.003,A -85,B 0,C 180,E1 -18342.71,E2 -18342.71} C_VEL
LIN {X 0,Y 148.638,Z 889.668,A -85,B 0,C 180,E1 -18344.992,E2 -18344.992} C_VEL
LIN {X 0,Y 140.937,Z 900.913,A -85,B 0,C 180,E1 -18351.459,E2 -18351.459} C_VEL
LIN {X 0,Y 140.014,Z 904.211,A -85,B 0,C 180,E1 -18353.795,E2 -18353.795} C_VEL
LIN {X 0,Y 140.5,Z 912.851,A -85,B 0,C 180,E1 -18360.814,E2 -18360.814} C_VEL
LIN {X 0,Y 143.071,Z 920.658,A -85,B 0,C 180,E1 -18368.843,E2 -18368.843} C_VEL
LIN {X 0,Y 148.351,Z 926.642,A -85,B 0,C 180,E1 -18376.846,E2 -18376.846} C_VEL
LIN {X 0,Y 156.764,Z 930.754,A -85,B 0,C 180,E1 -18384.491,E2 -18384.491} C_VEL
LIN {X 0,Y 168.461,Z 932.986,A -85,B 0,C 180,E1 -18391.486,E2 -18391.486} C_VEL
LIN {X 0,Y 176.244,Z 933.398,A -85,B 0,C 180,E1 -18394.958,E2 -18394.958} C_VEL
LIN {X 0,Y 156.134,Z 942.856,A -85,B 0,C 180,E1 -18405.215,E2 -18405.215} C_VEL
LIN {X 0,Y 144.112,Z 949.868,A -85,B 0,C 180,E1 -18416.761,E2 -18416.761} C_VEL
LIN {X 0,Y 139.17,Z 954.047,A -85,B 0,C 180,E1 -18427.617,E2 -18427.617} C_VEL
LIN {X 0,Y 138.489,Z 956.011,A -85,B 0,C 180,E1 -18437.071,E2 -18437.071} C_VEL
LIN {X 0,Y 138.919,Z 956.738,A -85,B 0,C 180,E1 -18441.305,E2 -18441.305} C_VEL
LIN {X 0,Y 139.737,Z 958.05,A -85,B 0,C 180,E1 -18447.538,E2 -18447.538} C_VEL
LIN {X 0,Y 139.813,Z 958.116,A -85,B 0,C 180,E1 -18451.638,E2 -18451.638} C_VEL
LIN {X 0,Y 139.152,Z 957.294,A -85,B 0,C 180,E1 -18456.6,E2 -18456.6} C_VEL
LIN {X 0,Y 138.526,Z 954.847,A -85,B 0,C 180,E1 -18463.353,E2 -18463.353} C_VEL
LIN {X 0,Y 139.18,Z 950.402,A -85,B 0,C 180,E1 -18471.05,E2 -18471.05} C_VEL
LIN {X 0,Y 141.75,Z 944.127,A -85,B 0,C 180,E1 -18478.661,E2 -18478.661} C_VEL
LIN {X 0,Y 146.398,Z 935.917,A -85,B 0,C 180,E1 -18485.968,E2 -18485.968} C_VEL
LIN {X 0,Y 152.661,Z 926.205,A -85,B 0,C 180,E1 -18492.422,E2 -18492.422} C_VEL
LIN {X 0,Y 160.324,Z 914.748,A -85,B 0,C 180,E1 -18498.142,E2 -18498.142} C_VEL
LIN {X 0,Y 168.248,Z 902.536,A -85,B 0,C 180,E1 -18502.78,E2 -18502.78} C_VEL
LIN {X 0,Y 176.817,Z 888.591,A -85,B 0,C 180,E1 -18506.813,E2 -18506.813} C_VEL
LIN {X 0,Y 185.124,Z 873.754,A -85,B 0,C 180,E1 -18510.095,E2 -18510.095} C_VEL
LIN {X 0,Y 192.838,Z 858.301,A -85,B 0,C 180,E1 -18512.713,E2 -18512.713} C_VEL
LIN {X 0,Y 200.276,Z 840.987,A -85,B 0,C 180,E1 -18514.973,E2 -18514.973} C_VEL
LIN {X 0,Y 206.769,Z 822.846,A -85,B 0,C 180,E1 -18516.745,E2 -18516.745} C_VEL
LIN {X 0,Y 212.133,Z 803.72,A -85,B 0,C 180,E1 -18518.114,E2 -18518.114} C_VEL
LIN {X 0,Y 216.065,Z 784.435,A -85,B 0,C 180,E1 -18519.073,E2 -18519.073} C_VEL
LIN {X 0,Y 218.432,Z 766.643,A -85,B 0,C 180,E1 -18519.647,E2 -18519.647} C_VEL
LIN {X 0,Y 221.447,Z 734.184,A -85,B 0,C 180,E1 -18520.498,E2 -18520.498} C_VEL
LIN {X 0,Y 223.353,Z 715.214,A -85,B 0,C 180,E1 -18520.897,E2 -18520.897} C_VEL
LIN {X 0,Y 229.769,Z 687.228,A -85,B 0,C 180,E1 -18521.63,E2 -18521.63} C_VEL
LIN {X 0,Y 231.064,Z 683.601,A -85,B 0,C 180,E1 -18521.77,E2 -18521.77} C_VEL
LIN {X 0,Y 242.812,Z 662.697,A -85,B 0,C 180,E1 -18522.899,E2 -18522.899} C_VEL
LIN {X 0,Y 244.42,Z 637.324,A -85,B 0,C 180,E1 -18527.119,E2 -18527.119} C_VEL
LIN {X 0,Y 249.001,Z 609.804,A -85,B 0,C 180,E1 -18531.224,E2 -18531.224} C_VEL
LIN {X 0,Y 249.354,Z 608.088,A -85,B 0,C 180,E1 -18531.469,E2 -18531.469} C_VEL
LIN {X 0,Y 242.42,Z 593.406,A -85,B 0,C 180,E1 -18536.454,E2 -18536.454} C_VEL
LIN {X 0,Y 235.734,Z 579.656,A -85,B 0,C 180,E1 -18541.702,E2 -18541.702} C_VEL
LIN {X 0,Y 229.299,Z 566.735,A -85,B 0,C 180,E1 -18547.265,E2 -18547.265} C_VEL
LIN {X 0,Y 230.595,Z 564.367,A -85,B 0,C 180,E1 -18549.233,E2 -18549.233} C_VEL
LIN {X 0,Y 231.749,Z 562.542,A -85,B 0,C 180,E1 -18550.692,E2 -18550.692} C_VEL
LIN {X 0,Y 233.986,Z 559.637,A -85,B 0,C 180,E1 -18553.09,E2 -18553.09} C_VEL
LIN {X 0,Y 238.256,Z 556.17,A -85,B 0,C 180,E1 -18556.833,E2 -18556.833} C_VEL
LIN {X 0,Y 244.351,Z 553.406,A -85,B 0,C 180,E1 -18561.043,E2 -18561.043} C_VEL
LIN {X 0,Y 246.077,Z 558.169,A -85,B 0,C 180,E1 -18562.494,E2 -18562.494} C_VEL
LIN {X 0,Y 231.033,Z 720.141,A -85,B 0,C 180,E1 -18566.19,E2 -18566.19} C_VEL
LIN {X 0,Y 228.58,Z 749.113,A -85,B 0,C 180,E1 -18567.177,E2 -18567.177} C_VEL
LIN {X 0,Y 225.59,Z 767.906,A -85,B 0,C 180,E1 -18568.15,E2 -18568.15} C_VEL
LIN {X 0,Y 221.444,Z 785.453,A -85,B 0,C 180,E1 -18569.376,E2 -18569.376} C_VEL
LIN {X 0,Y 216.178,Z 802.196,A -85,B 0,C 180,E1 -18570.891,E2 -18570.891} C_VEL
LIN {X 0,Y 209.713,Z 818.623,A -85,B 0,C 180,E1 -18572.812,E2 -18572.812} C_VEL
LIN {X 0,Y 202.359,Z 834.094,A -85,B 0,C 180,E1 -18575.142,E2 -18575.142} C_VEL
LIN {X 0,Y 194.098,Z 848.785,A -85,B 0,C 180,E1 -18577.988,E2 -18577.988} C_VEL
LIN {X 0,Y 185.297,Z 862.323,A -85,B 0,C 180,E1 -18581.407,E2 -18581.407} C_VEL
LIN {X 0,Y 176.505,Z 874.256,A -85,B 0,C 180,E1 -18585.379,E2 -18585.379} C_VEL
LIN {X 0,Y 167.951,Z 884.673,A -85,B 0,C 180,E1 -18589.989,E2 -18589.989} C_VEL
LIN {X 0,Y 159.962,Z 893.588,A -85,B 0,C 180,E1 -18595.334,E2 -18595.334} C_VEL
LIN {X 0,Y 152.9,Z 900.971,A -85,B 0,C 180,E1 -18601.487,E2 -18601.487} C_VEL
LIN {X 0,Y 147.118,Z 906.724,A -85,B 0,C 180,E1 -18608.47,E2 -18608.47} C_VEL
LIN {X 0,Y 143.186,Z 910.603,A -85,B 0,C 180,E1 -18615.855,E2 -18615.855} C_VEL
LIN {X 0,Y 141.044,Z 912.772,A -85,B 0,C 180,E1 -18623.488,E2 -18623.488} C_VEL
LIN {X 0,Y 140.509,Z 913.35,A -85,B 0,C 180,E1 -18630.817,E2 -18630.817} C_VEL
LIN {X 0,Y 141.348,Z 912.505,A -85,B 0,C 180,E1 -18638.134,E2 -18638.134} C_VEL
LIN {X 0,Y 143.829,Z 910.008,A -85,B 0,C 180,E1 -18645.732,E2 -18645.732} C_VEL
LIN {X 0,Y 148.13,Z 905.762,A -85,B 0,C 180,E1 -18653.049,E2 -18653.049} C_VEL
LIN {X 0,Y 153.904,Z 899.995,A -85,B 0,C 180,E1 -18659.588,E2 -18659.588} C_VEL
LIN {X 0,Y 161.207,Z 892.34,A -85,B 0,C 180,E1 -18665.665,E2 -18665.665} C_VEL
LIN {X 0,Y 169.402,Z 883.121,A -85,B 0,C 180,E1 -18670.933,E2 -18670.933} C_VEL
LIN {X 0,Y 178.121,Z 872.361,A -85,B 0,C 180,E1 -18675.472,E2 -18675.472} C_VEL
LIN {X 0,Y 186.444,Z 860.903,A -85,B 0,C 180,E1 -18679.135,E2 -18679.135} C_VEL
LIN {X 0,Y 187.587,Z 859.126,A -85,B 0,C 180,E1 -18679.69,E2 -18679.69} C_VEL
LIN {X 0,Y 180.024,Z 862.534,A -85,B 0,C 180,E1 -18681.533,E2 -18681.533} C_VEL
LIN {X 0,Y 170.317,Z 866.759,A -85,B 0,C 180,E1 -18684.465,E2 -18684.465} C_VEL
LIN {X 0,Y 162.239,Z 870.178,A -85,B 0,C 180,E1 -18687.576,E2 -18687.576} C_VEL
LIN {X 0,Y 155.543,Z 872.994,A -85,B 0,C 180,E1 -18690.754,E2 -18690.754} C_VEL
LIN {X 0,Y 153.374,Z 873.87,A -85,B 0,C 180,E1 -18692.005,E2 -18692.005} C_VEL
LIN {X 0,Y 149.685,Z 875.476,A -85,B 0,C 180,E1 -18694.265,E2 -18694.265} C_VEL
LIN {X 0,Y 148.396,Z 875.963,A -85,B 0,C 180,E1 -18695.307,E2 -18695.307} C_VEL
LIN {X 0,Y 145.419,Z 877.436,A -85,B 0,C 180,E1 -18697.353,E2 -18697.353} C_VEL
LIN {X 0,Y 144.202,Z 877.925,A -85,B 0,C 180,E1 -18698.865,E2 -18698.865} C_VEL
LIN {X 0,Y 141.621,Z 890.126,A -85,B 0,C 180,E1 -18704.856,E2 -18704.856} C_VEL
LIN {X 0,Y 140.154,Z 901.428,A -85,B 0,C 180,E1 -18711.796,E2 -18711.796} C_VEL
LIN {X 0,Y 140.014,Z 904.211,A -85,B 0,C 180,E1 -18713.795,E2 -18713.795} C_VEL
LIN {X 0,Y 139.024,Z 907.881,A -85,B 0,C 180,E1 -18716.575,E2 -18716.575} C_VEL
LIN {X 0,Y 134.061,Z 916.581,A -85,B 0,C 180,E1 -18724.468,E2 -18724.468} C_VEL
LIN {X 0,Y 134.212,Z 919.059,A -85,B 0,C 180,E1 -18727.119,E2 -18727.119} C_VEL
LIN {X 0,Y 138.573,Z 925.538,A -85,B 0,C 180,E1 -18735.054,E2 -18735.054} C_VEL
LIN {X 0,Y 146.045,Z 930.607,A -85,B 0,C 180,E1 -18742.968,E2 -18742.968} C_VEL
LIN {X 0,Y 156.737,Z 933.958,A -85,B 0,C 180,E1 -18750.261,E2 -18750.261} C_VEL
LIN {X 0,Y 165.966,Z 935.305,A -85,B 0,C 180,E1 -18754.891,E2 -18754.891} C_VEL
LIN {X 0,Y 146.227,Z 943.749,A -85,B 0,C 180,E1 -18765.885,E2 -18765.885} C_VEL
LIN {X 0,Y 134.959,Z 949.715,A -85,B 0,C 180,E1 -18778.262,E2 -18778.262} C_VEL
LIN {X 0,Y 130.882,Z 953.067,A -85,B 0,C 180,E1 -18789.989,E2 -18789.989} C_VEL
LIN {X 0,Y 130.711,Z 954.369,A -85,B 0,C 180,E1 -18797.631,E2 -18797.631} C_VEL
LIN {X 0,Y 131.438,Z 956.402,A -85,B 0,C 180,E1 -18804.761,E2 -18804.761} C_VEL
LIN {X 0,Y 131.979,Z 956.955,A -85,B 0,C 180,E1 -18809.803,E2 -18809.803} C_VEL
LIN {X 0,Y 131.491,Z 956.481,A -85,B 0,C 180,E1 -18814.797,E2 -18814.797} C_VEL
LIN {X 0,Y 130.663,Z 954.595,A -85,B 0,C 180,E1 -18821.633,E2 -18821.633} C_VEL
LIN {X 0,Y 130.933,Z 950.775,A -85,B 0,C 180,E1 -18829.632,E2 -18829.632} C_VEL
LIN {X 0,Y 133.208,Z 945.107,A -85,B 0,C 180,E1 -18837.733,E2 -18837.733} C_VEL
LIN {X 0,Y 137.745,Z 937.456,A -85,B 0,C 180,E1 -18845.614,E2 -18845.614} C_VEL
LIN {X 0,Y 144.318,Z 927.973,A -85,B 0,C 180,E1 -18852.761,E2 -18852.761} C_VEL
LIN {X 0,Y 152.43,Z 916.731,A -85,B 0,C 180,E1 -18858.966,E2 -18858.966} C_VEL
LIN {X 0,Y 160.847,Z 904.776,A -85,B 0,C 180,E1 -18863.91,E2 -18863.91} C_VEL
LIN {X 0,Y 170.006,Z 890.971,A -85,B 0,C 180,E1 -18868.194,E2 -18868.194} C_VEL
LIN {X 0,Y 178.992,Z 876.145,A -85,B 0,C 180,E1 -18871.654,E2 -18871.654} C_VEL
LIN {X 0,Y 187.348,Z 860.618,A -85,B 0,C 180,E1 -18874.412,E2 -18874.412} C_VEL
LIN {X 0,Y 194.966,Z 844.273,A -85,B 0,C 180,E1 -18876.63,E2 -18876.63} C_VEL
LIN {X 0,Y 201.675,Z 827.275,A -85,B 0,C 180,E1 -18878.368,E2 -18878.368} C_VEL
LIN {X 0,Y 207.111,Z 810.438,A -85,B 0,C 180,E1 -18879.661,E2 -18879.661} C_VEL
LIN {X 0,Y 211.14,Z 794.583,A -85,B 0,C 180,E1 -18880.578,E2 -18880.578} C_VEL
LIN {X 0,Y 214.123,Z 778.377,A -85,B 0,C 180,E1 -18881.253,E2 -18881.253} C_VEL
LIN {X 0,Y 216.938,Z 753.324,A -85,B 0,C 180,E1 -18881.962,E2 -18881.962} C_VEL
LIN {X 0,Y 218.956,Z 732.025,A -85,B 0,C 180,E1 -18882.534,E2 -18882.534} C_VEL
LIN {X 0,Y 222.206,Z 701.843,A -85,B 0,C 180,E1 -18883.043,E2 -18883.043} C_VEL
LIN {X 0,Y 224.7,Z 683.974,A -85,B 0,C 180,E1 -18883.075,E2 -18883.075} C_VEL
LIN {X 0,Y 236.447,Z 663.172,A -85,B 0,C 180,E1 -18884.236,E2 -18884.236} C_VEL
LIN {X 0,Y 238.513,Z 637.656,A -85,B 0,C 180,E1 -18888.515,E2 -18888.515} C_VEL
LIN {X 0,Y 243.017,Z 611.87,A -85,B 0,C 180,E1 -18892.435,E2 -18892.435} C_VEL
LIN {X 0,Y 236.69,Z 598.398,A -85,B 0,C 180,E1 -18897.095,E2 -18897.095} C_VEL
LIN {X 0,Y 229.954,Z 584.486,A -85,B 0,C 180,E1 -18902.493,E2 -18902.493} C_VEL
LIN {X 0,Y 227.049,Z 578.552,A -85,B 0,C 180,E1 -18905.054,E2 -18905.054} C_VEL
LIN {X 0,Y 228.356,Z 575.16,A -85,B 0,C 180,E1 -18907.485,E2 -18907.485} C_VEL
LIN {X 0,Y 229.211,Z 573.479,A -85,B 0,C 180,E1 -18908.783,E2 -18908.783} C_VEL
LIN {X 0,Y 231.064,Z 570.358,A -85,B 0,C 180,E1 -18911.103,E2 -18911.103} C_VEL
LIN {X 0,Y 234.529,Z 566.243,A -85,B 0,C 180,E1 -18914.569,E2 -18914.569} C_VEL
LIN {X 0,Y 241.431,Z 562.145,A -85,B 0,C 180,E1 -18919.853,E2 -18919.853} C_VEL
LIN {X 0,Y 242.722,Z 561.674,A -85,B 0,C 180,E1 -18920.686,E2 -18920.686} C_VEL
LIN {X 0,Y 242.834,Z 562.472,A -85,B 0,C 180,E1 -18920.828,E2 -18920.828} C_VEL
LIN {X 0,Y 227.694,Z 720.669,A -85,B 0,C 180,E1 -18924.378,E2 -18924.378} C_VEL
LIN {X 0,Y 225.074,Z 750.318,A -85,B 0,C 180,E1 -18925.384,E2 -18925.384} C_VEL
LIN {X 0,Y 221.991,Z 769.031,A -85,B 0,C 180,E1 -18926.343,E2 -18926.343} C_VEL
LIN {X 0,Y 217.675,Z 786.693,A -85,B 0,C 180,E1 -18927.562,E2 -18927.562} C_VEL
LIN {X 0,Y 212.236,Z 803.426,A -85,B 0,C 180,E1 -18929.058,E2 -18929.058} C_VEL
LIN {X 0,Y 205.78,Z 819.354,A -85,B 0,C 180,E1 -18930.891,E2 -18930.891} C_VEL
LIN {X 0,Y 198.266,Z 834.711,A -85,B 0,C 180,E1 -18933.162,E2 -18933.162} C_VEL
LIN {X 0,Y 190.009,Z 848.983,A -85,B 0,C 180,E1 -18935.869,E2 -18935.869} C_VEL
LIN {X 0,Y 181.442,Z 861.818,A -85,B 0,C 180,E1 -18939.015,E2 -18939.015} C_VEL
LIN {X 0,Y 172.745,Z 873.323,A -85,B 0,C 180,E1 -18942.687,E2 -18942.687} C_VEL
LIN {X 0,Y 163.58,Z 884.135,A -85,B 0,C 180,E1 -18947.277,E2 -18947.277} C_VEL
LIN {X 0,Y 154.909,Z 893.403,A -85,B 0,C 180,E1 -18952.648,E2 -18952.648} C_VEL
LIN {X 0,Y 147.12,Z 901.108,A -85,B 0,C 180,E1 -18958.908,E2 -18958.908} C_VEL
LIN {X 0,Y 140.92,Z 906.911,A -85,B 0,C 180,E1 -18965.701,E2 -18965.701} C_VEL
LIN {X 0,Y 136.254,Z 911.191,A -85,B 0,C 180,E1 -18973.371,E2 -18973.371} C_VEL
LIN {X 0,Y 133.541,Z 913.723,A -85,B 0,C 180,E1 -18981.389,E2 -18981.389} C_VEL
LIN {X 0,Y 132.608,Z 914.626,A -85,B 0,C 180,E1 -18989.569,E2 -18989.569} C_VEL
LIN {X 0,Y 133.347,Z 913.943,A -85,B 0,C 180,E1 -18997.758,E2 -18997.758} C_VEL
LIN {X 0,Y 135.854,Z 911.642,A -85,B 0,C 180,E1 -19005.803,E2 -19005.803} C_VEL
LIN {X 0,Y 140.295,Z 907.589,A -85,B 0,C 180,E1 -19013.523,E2 -19013.523} C_VEL
LIN {X 0,Y 146.678,Z 901.638,A -85,B 0,C 180,E1 -19020.748,E2 -19020.748} C_VEL
LIN {X 0,Y 153.902,Z 894.572,A -85,B 0,C 180,E1 -19026.707,E2 -19026.707} C_VEL
LIN {X 0,Y 162.42,Z 885.585,A -85,B 0,C 180,E1 -19032.146,E2 -19032.146} C_VEL
LIN {X 0,Y 171.469,Z 875.084,A -85,B 0,C 180,E1 -19036.795,E2 -19036.795} C_VEL
LIN {X 0,Y 177.687,Z 867.161,A -85,B 0,C 180,E1 -19039.558,E2 -19039.558} C_VEL
LIN {X 0,Y 167.359,Z 871.398,A -85,B 0,C 180,E1 -19042.454,E2 -19042.454} C_VEL
LIN {X 0,Y 158.248,Z 875.002,A -85,B 0,C 180,E1 -19045.782,E2 -19045.782} C_VEL
LIN {X 0,Y 150.706,Z 877.997,A -85,B 0,C 180,E1 -19049.278,E2 -19049.278} C_VEL
LIN {X 0,Y 144.59,Z 880.455,A -85,B 0,C 180,E1 -19052.844,E2 -19052.844} C_VEL
LIN {X 0,Y 142.554,Z 881.307,A -85,B 0,C 180,E1 -19054.222,E2 -19054.222} C_VEL
LIN {X 0,Y 139.353,Z 882.669,A -85,B 0,C 180,E1 -19056.756,E2 -19056.756} C_VEL
LIN {X 0,Y 138.092,Z 883.232,A -85,B 0,C 180,E1 -19057.881,E2 -19057.881} C_VEL
LIN {X 0,Y 135.297,Z 884.6,A -85,B 0,C 180,E1 -19060.575,E2 -19060.575} C_VEL
LIN {X 0,Y 134.735,Z 884.9,A -85,B 0,C 180,E1 -19061.614,E2 -19061.614} C_VEL
LIN {X 0,Y 132.769,Z 895.791,A -85,B 0,C 180,E1 -19067.826,E2 -19067.826} C_VEL
LIN {X 0,Y 131.994,Z 906.795,A -85,B 0,C 180,E1 -19075.654,E2 -19075.654} C_VEL
LIN {X 0,Y 133.035,Z 915.52,A -85,B 0,C 180,E1 -19083.446,E2 -19083.446} C_VEL
LIN {X 0,Y 134.212,Z 919.059,A -85,B 0,C 180,E1 -19087.119,E2 -19087.119} C_VEL
LIN {X 0,Y 134.589,Z 921.798,A -85,B 0,C 180,E1 -19090.214,E2 -19090.214} C_VEL
LIN {X 0,Y 133.935,Z 928.049,A -85,B 0,C 180,E1 -19098.638,E2 -19098.638} C_VEL
LIN {X 0,Y 135.716,Z 929.899,A -85,B 0,C 180,E1 -19101.502,E2 -19101.502} C_VEL
LIN {X 0,Y 145.068,Z 934.078,A -85,B 0,C 180,E1 -19108.845,E2 -19108.845} C_VEL
LIN {X 0,Y 155.825,Z 936.573,A -85,B 0,C 180,E1 -19114.781,E2 -19114.781} C_VEL
LIN {X 0,Y 136.575,Z 944.004,A -85,B 0,C 180,E1 -19126.513,E2 -19126.513} C_VEL
LIN {X 0,Y 125.968,Z 949.124,A -85,B 0,C 180,E1 -19139.995,E2 -19139.995} C_VEL
LIN {X 0,Y 122.905,Z 951.574,A -85,B 0,C 180,E1 -19152.138,E2 -19152.138} C_VEL
LIN {X 0,Y 122.742,Z 952.486,A -85,B 0,C 180,E1 -19155.372,E2 -19155.372} C_VEL
LIN {X 0,Y 123.324,Z 954.929,A -85,B 0,C 180,E1 -19163.481,E2 -19163.481} C_VEL
LIN {X 0,Y 124.015,Z 955.62,A -85,B 0,C 180,E1 -19168.624,E2 -19168.624} C_VEL
LIN {X 0,Y 123.873,Z 955.507,A -85,B 0,C 180,E1 -19172.775,E2 -19172.775} C_VEL
LIN {X 0,Y 122.871,Z 954.095,A -85,B 0,C 180,E1 -19179.838,E2 -19179.838} C_VEL
LIN {X 0,Y 122.768,Z 950.956,A -85,B 0,C 180,E1 -19188.027,E2 -19188.027} C_VEL
LIN {X 0,Y 124.695,Z 945.88,A -85,B 0,C 180,E1 -19196.68,E2 -19196.68} C_VEL
LIN {X 0,Y 128.957,Z 938.948,A -85,B 0,C 180,E1 -19205.011,E2 -19205.011} C_VEL
LIN {X 0,Y 135.546,Z 930.028,A -85,B 0,C 180,E1 -19212.736,E2 -19212.736} C_VEL
LIN {X 0,Y 143.716,Z 919.568,A -85,B 0,C 180,E1 -19219.316,E2 -19219.316} C_VEL
LIN {X 0,Y 153.059,Z 907.398,A -85,B 0,C 180,E1 -19224.911,E2 -19224.911} C_VEL
LIN {X 0,Y 162.955,Z 893.665,A -85,B 0,C 180,E1 -19229.549,E2 -19229.549} C_VEL
LIN {X 0,Y 172.552,Z 879.116,A -85,B 0,C 180,E1 -19233.169,E2 -19233.169} C_VEL
LIN {X 0,Y 181.174,Z 864.334,A -85,B 0,C 180,E1 -19235.971,E2 -19235.971} C_VEL
LIN {X 0,Y 189.43,Z 848.202,A -85,B 0,C 180,E1 -19238.273,E2 -19238.273} C_VEL
LIN {X 0,Y 196.749,Z 831.373,A -85,B 0,C 180,E1 -19240.075,E2 -19240.075} C_VEL
LIN {X 0,Y 202.535,Z 815.151,A -85,B 0,C 180,E1 -19241.412,E2 -19241.412} C_VEL
LIN {X 0,Y 207.535,Z 797.447,A -85,B 0,C 180,E1 -19242.498,E2 -19242.498} C_VEL
LIN {X 0,Y 211.267,Z 779.43,A -85,B 0,C 180,E1 -19243.259,E2 -19243.259} C_VEL
LIN {X 0,Y 214.082,Z 757.251,A -85,B 0,C 180,E1 -19243.872,E2 -19243.872} C_VEL
LIN {X 0,Y 217.927,Z 718.944,A -85,B 0,C 180,E1 -19244.808,E2 -19244.808} C_VEL
LIN {X 0,Y 221.202,Z 691.094,A -85,B 0,C 180,E1 -19245.061,E2 -19245.061} C_VEL
LIN {X 0,Y 223.253,Z 675.543,A -85,B 0,C 180,E1 -19245,E2 -19245} C_VEL
LIN {X 0,Y 230.16,Z 663.524,A -85,B 0,C 180,E1 -19245.637,E2 -19245.637} C_VEL
LIN {X 0,Y 232.69,Z 637.904,A -85,B 0,C 180,E1 -19249.966,E2 -19249.966} C_VEL
LIN {X 0,Y 236.76,Z 615.907,A -85,B 0,C 180,E1 -19253.332,E2 -19253.332} C_VEL
LIN {X 0,Y 230.324,Z 602.039,A -85,B 0,C 180,E1 -19258.259,E2 -19258.259} C_VEL
LIN {X 0,Y 225.061,Z 590.926,A -85,B 0,C 180,E1 -19262.674,E2 -19262.674} C_VEL
LIN {X 0,Y 226.066,Z 587.04,A -85,B 0,C 180,E1 -19265.266,E2 -19265.266} C_VEL
LIN {X 0,Y 226.892,Z 584.763,A -85,B 0,C 180,E1 -19266.834,E2 -19266.834} C_VEL
LIN {X 0,Y 228.383,Z 581.441,A -85,B 0,C 180,E1 -19269.069,E2 -19269.069} C_VEL
LIN {X 0,Y 232.522,Z 575.475,A -85,B 0,C 180,E1 -19273.681,E2 -19273.681} C_VEL
LIN {X 0,Y 237.264,Z 571.77,A -85,B 0,C 180,E1 -19277.664,E2 -19277.664} C_VEL
LIN {X 0,Y 239.396,Z 570.79,A -85,B 0,C 180,E1 -19279.201,E2 -19279.201} C_VEL
LIN {X 0,Y 224.587,Z 721.223,A -85,B 0,C 180,E1 -19282.516,E2 -19282.516} C_VEL
LIN {X 0,Y 221.795,Z 751.523,A -85,B 0,C 180,E1 -19283.536,E2 -19283.536} C_VEL
LIN {X 0,Y 218.595,Z 770.259,A -85,B 0,C 180,E1 -19284.484,E2 -19284.484} C_VEL
LIN {X 0,Y 214.132,Z 787.933,A -85,B 0,C 180,E1 -19285.687,E2 -19285.687} C_VEL
LIN {X 0,Y 208.474,Z 804.769,A -85,B 0,C 180,E1 -19287.169,E2 -19287.169} C_VEL
LIN {X 0,Y 201.75,Z 820.787,A -85,B 0,C 180,E1 -19288.99,E2 -19288.99} C_VEL
LIN {X 0,Y 194.056,Z 835.966,A -85,B 0,C 180,E1 -19291.208,E2 -19291.208} C_VEL
LIN {X 0,Y 185.487,Z 850.242,A -85,B 0,C 180,E1 -19293.889,E2 -19293.889} C_VEL
LIN {X 0,Y 176.569,Z 863.08,A -85,B 0,C 180,E1 -19297.02,E2 -19297.02} C_VEL
LIN {X 0,Y 167.479,Z 874.587,A -85,B 0,C 180,E1 -19300.696,E2 -19300.696} C_VEL
LIN {X 0,Y 157.853,Z 885.401,A -85,B 0,C 180,E1 -19305.326,E2 -19305.326} C_VEL
LIN {X 0,Y 148.688,Z 894.669,A -85,B 0,C 180,E1 -19310.796,E2 -19310.796} C_VEL
LIN {X 0,Y 140.397,Z 902.371,A -85,B 0,C 180,E1 -19317.233,E2 -19317.233} C_VEL
LIN {X 0,Y 133.739,Z 908.178,A -85,B 0,C 180,E1 -19324.304,E2 -19324.304} C_VEL
LIN {X 0,Y 128.688,Z 912.458,A -85,B 0,C 180,E1 -19332.363,E2 -19332.363} C_VEL
LIN {X 0,Y 125.729,Z 914.988,A -85,B 0,C 180,E1 -19340.85,E2 -19340.85} C_VEL
LIN {X 0,Y 124.708,Z 915.889,A -85,B 0,C 180,E1 -19349.542,E2 -19349.542} C_VEL
LIN {X 0,Y 125.519,Z 915.207,A -85,B 0,C 180,E1 -19358.245,E2 -19358.245} C_VEL
LIN {X 0,Y 128.255,Z 912.907,A -85,B 0,C 180,E1 -19366.766,E2 -19366.766} C_VEL
LIN {X 0,Y 133.068,Z 908.855,A -85,B 0,C 180,E1 -19374.885,E2 -19374.885} C_VEL
LIN {X 0,Y 139.924,Z 902.903,A -85,B 0,C 180,E1 -19382.408,E2 -19382.408} C_VEL
LIN {X 0,Y 147.623,Z 895.836,A -85,B 0,C 180,E1 -19388.546,E2 -19388.546} C_VEL
LIN {X 0,Y 156.637,Z 886.846,A -85,B 0,C 180,E1 -19394.091,E2 -19394.091} C_VEL
LIN {X 0,Y 166.149,Z 876.343,A -85,B 0,C 180,E1 -19398.786,E2 -19398.786} C_VEL
LIN {X 0,Y 167.594,Z 874.639,A -85,B 0,C 180,E1 -19399.435,E2 -19399.435} C_VEL
LIN {X 0,Y 154.28,Z 879.582,A -85,B 0,C 180,E1 -19403.859,E2 -19403.859} C_VEL
LIN {X 0,Y 146.367,Z 882.538,A -85,B 0,C 180,E1 -19407.338,E2 -19407.338} C_VEL
LIN {X 0,Y 139.417,Z 885.177,A -85,B 0,C 180,E1 -19411.28,E2 -19411.28} C_VEL
LIN {X 0,Y 133.905,Z 887.388,A -85,B 0,C 180,E1 -19415.281,E2 -19415.281} C_VEL
LIN {X 0,Y 129.604,Z 889.306,A -85,B 0,C 180,E1 -19419.213,E2 -19419.213} C_VEL
LIN {X 0,Y 128.16,Z 890.001,A -85,B 0,C 180,E1 -19420.871,E2 -19420.871} C_VEL
LIN {X 0,Y 125.855,Z 891.248,A -85,B 0,C 180,E1 -19423.854,E2 -19423.854} C_VEL
LIN {X 0,Y 125.445,Z 891.691,A -85,B 0,C 180,E1 -19424.985,E2 -19424.985} C_VEL
LIN {X 0,Y 124.094,Z 902.543,A -85,B 0,C 180,E1 -19432.336,E2 -19432.336} C_VEL
LIN {X 0,Y 124.474,Z 912.732,A -85,B 0,C 180,E1 -19440.919,E2 -19440.919} C_VEL
LIN {X 0,Y 127.296,Z 921.33,A -85,B 0,C 180,E1 -19449.949,E2 -19449.949} C_VEL
LIN {X 0,Y 133.186,Z 928.145,A -85,B 0,C 180,E1 -19458.832,E2 -19458.832} C_VEL
LIN {X 0,Y 135.716,Z 929.899,A -85,B 0,C 180,E1 -19461.502,E2 -19461.502} C_VEL
LIN {X 0,Y 136.878,Z 931.217,A -85,B 0,C 180,E1 -19463.58,E2 -19463.58} C_VEL
LIN {X 0,Y 137.566,Z 934.655,A -85,B 0,C 180,E1 -19469.445,E2 -19469.445} C_VEL
LIN {X 0,Y 139.284,Z 935.582,A -85,B 0,C 180,E1 -19471.116,E2 -19471.116} C_VEL
LIN {X 0,Y 145.636,Z 937.361,A -85,B 0,C 180,E1 -19474.717,E2 -19474.717} C_VEL
LIN {X 0,Y 126.92,Z 943.853,A -85,B 0,C 180,E1 -19487.35,E2 -19487.35} C_VEL
LIN {X 0,Y 117.349,Z 947.95,A -85,B 0,C 180,E1 -19501.499,E2 -19501.499} C_VEL
LIN {X 0,Y 115.259,Z 949.484,A -85,B 0,C 180,E1 -19510.224,E2 -19510.224} C_VEL
LIN {X 0,Y 114.941,Z 952.826,A -85,B 0,C 180,E1 -19519.473,E2 -19519.473} C_VEL
LIN {X 0,Y 115.938,Z 954.241,A -85,B 0,C 180,E1 -19527.033,E2 -19527.033} C_VEL
LIN {X 0,Y 116.101,Z 954.349,A -85,B 0,C 180,E1 -19531.479,E2 -19531.479} C_VEL
LIN {X 0,Y 115.224,Z 953.525,A -85,B 0,C 180,E1 -19537.478,E2 -19537.478} C_VEL
LIN {X 0,Y 114.701,Z 950.907,A -85,B 0,C 180,E1 -19546.196,E2 -19546.196} C_VEL
LIN {X 0,Y 116.381,Z 946.106,A -85,B 0,C 180,E1 -19555.985,E2 -19555.985} C_VEL
LIN {X 0,Y 120.542,Z 939.692,A -85,B 0,C 180,E1 -19564.912,E2 -19564.912} C_VEL
LIN {X 0,Y 127.199,Z 931.355,A -85,B 0,C 180,E1 -19573.145,E2 -19573.145} C_VEL
LIN {X 0,Y 135.552,Z 921.522,A -85,B 0,C 180,E1 -19580.095,E2 -19580.095} C_VEL
LIN {X 0,Y 144.987,Z 910.265,A -85,B 0,C 180,E1 -19585.845,E2 -19585.845} C_VEL
LIN {X 0,Y 155.148,Z 897.339,A -85,B 0,C 180,E1 -19590.675,E2 -19590.675} C_VEL
LIN {X 0,Y 165.142,Z 883.517,A -85,B 0,C 180,E1 -19594.437,E2 -19594.437} C_VEL
LIN {X 0,Y 175.146,Z 867.833,A -85,B 0,C 180,E1 -19597.638,E2 -19597.638} C_VEL
LIN {X 0,Y 184.463,Z 851.047,A -85,B 0,C 180,E1 -19600.123,E2 -19600.123} C_VEL
LIN {X 0,Y 191.975,Z 835.168,A -85,B 0,C 180,E1 -19601.896,E2 -19601.896} C_VEL
LIN {X 0,Y 198.772,Z 817.734,A -85,B 0,C 180,E1 -19603.382,E2 -19603.382} C_VEL
LIN {X 0,Y 204.473,Z 799.163,A -85,B 0,C 180,E1 -19604.529,E2 -19604.529} C_VEL
LIN {X 0,Y 208.712,Z 780.292,A -85,B 0,C 180,E1 -19605.322,E2 -19605.322} C_VEL
LIN {X 0,Y 211.463,Z 761.346,A -85,B 0,C 180,E1 -19605.815,E2 -19605.815} C_VEL
LIN {X 0,Y 215.714,Z 719.942,A -85,B 0,C 180,E1 -19606.837,E2 -19606.837} C_VEL
LIN {X 0,Y 219.13,Z 691.134,A -85,B 0,C 180,E1 -19607.074,E2 -19607.074} C_VEL
LIN {X 0,Y 222.037,Z 668.964,A -85,B 0,C 180,E1 -19606.965,E2 -19606.965} C_VEL
LIN {X 0,Y 222.751,Z 666.103,A -85,B 0,C 180,E1 -19606.914,E2 -19606.914} C_VEL
LIN {X 0,Y 223.883,Z 664.081,A -85,B 0,C 180,E1 -19607.026,E2 -19607.026} C_VEL
LIN {X 0,Y 226.955,Z 637.717,A -85,B 0,C 180,E1 -19611.514,E2 -19611.514} C_VEL
LIN {X 0,Y 230.514,Z 619.887,A -85,B 0,C 180,E1 -19614.275,E2 -19614.275} C_VEL
LIN {X 0,Y 224.563,Z 606.945,A -85,B 0,C 180,E1 -19618.98,E2 -19618.98} C_VEL
LIN {X 0,Y 223.369,Z 604.16,A -85,B 0,C 180,E1 -19620.129,E2 -19620.129} C_VEL
LIN {X 0,Y 224.055,Z 599.384,A -85,B 0,C 180,E1 -19622.942,E2 -19622.942} C_VEL
LIN {X 0,Y 224.575,Z 597.202,A -85,B 0,C 180,E1 -19624.341,E2 -19624.341} C_VEL
LIN {X 0,Y 226.091,Z 592.623,A -85,B 0,C 180,E1 -19627.241,E2 -19627.241} C_VEL
LIN {X 0,Y 228.021,Z 588.707,A -85,B 0,C 180,E1 -19629.975,E2 -19629.975} C_VEL
LIN {X 0,Y 232.054,Z 583.163,A -85,B 0,C 180,E1 -19634.218,E2 -19634.218} C_VEL
LIN {X 0,Y 236.059,Z 580.065,A -85,B 0,C 180,E1 -19637.548,E2 -19637.548} C_VEL
LIN {X 0,Y 221.734,Z 721.674,A -85,B 0,C 180,E1 -19640.6,E2 -19640.6} C_VEL
LIN {X 0,Y 218.753,Z 752.728,A -85,B 0,C 180,E1 -19641.634,E2 -19641.634} C_VEL
LIN {X 0,Y 215.438,Z 771.488,A -85,B 0,C 180,E1 -19642.57,E2 -19642.57} C_VEL
LIN {X 0,Y 210.826,Z 789.174,A -85,B 0,C 180,E1 -19643.751,E2 -19643.751} C_VEL
LIN {X 0,Y 204.987,Z 806.017,A -85,B 0,C 180,E1 -19645.204,E2 -19645.204} C_VEL
LIN {X 0,Y 198.041,Z 822.04,A -85,B 0,C 180,E1 -19646.99,E2 -19646.99} C_VEL
LIN {X 0,Y 190.081,Z 837.222,A -85,B 0,C 180,E1 -19649.17,E2 -19649.17} C_VEL
LIN {X 0,Y 181.197,Z 851.501,A -85,B 0,C 180,E1 -19651.814,E2 -19651.814} C_VEL
LIN {X 0,Y 171.922,Z 864.341,A -85,B 0,C 180,E1 -19654.915,E2 -19654.915} C_VEL
LIN {X 0,Y 162.429,Z 875.851,A -85,B 0,C 180,E1 -19658.579,E2 -19658.579} C_VEL
LIN {X 0,Y 152.323,Z 886.666,A -85,B 0,C 180,E1 -19663.231,E2 -19663.231} C_VEL
LIN {X 0,Y 142.636,Z 895.936,A -85,B 0,C 180,E1 -19668.783,E2 -19668.783} C_VEL
LIN {X 0,Y 133.802,Z 903.638,A -85,B 0,C 180,E1 -19675.396,E2 -19675.396} C_VEL
LIN {X 0,Y 126.647,Z 909.445,A -85,B 0,C 180,E1 -19682.75,E2 -19682.75} C_VEL
LIN {X 0,Y 121.167,Z 913.724,A -85,B 0,C 180,E1 -19691.228,E2 -19691.228} C_VEL
LIN {X 0,Y 117.93,Z 916.253,A -85,B 0,C 180,E1 -19700.239,E2 -19700.239} C_VEL
LIN {X 0,Y 116.809,Z 917.152,A -85,B 0,C 180,E1 -19709.511,E2 -19709.511} C_VEL
LIN {X 0,Y 117.7,Z 916.471,A -85,B 0,C 180,E1 -19718.797,E2 -19718.797} C_VEL
LIN {X 0,Y 120.696,Z 914.172,A -85,B 0,C 180,E1 -19727.851,E2 -19727.851} C_VEL
LIN {X 0,Y 125.923,Z 910.12,A -85,B 0,C 180,E1 -19736.403,E2 -19736.403} C_VEL
LIN {X 0,Y 132.865,Z 904.547,A -85,B 0,C 180,E1 -19743.842,E2 -19743.842} C_VEL
LIN {X 0,Y 141.511,Z 897.099,A -85,B 0,C 180,E1 -19750.546,E2 -19750.546} C_VEL
LIN {X 0,Y 151.048,Z 888.108,A -85,B 0,C 180,E1 -19756.182,E2 -19756.182} C_VEL
LIN {X 0,Y 157.548,Z 881.389,A -85,B 0,C 180,E1 -19759.395,E2 -19759.395} C_VEL
LIN {X 0,Y 149.681,Z 884.136,A -85,B 0,C 180,E1 -19762.079,E2 -19762.079} C_VEL
LIN {X 0,Y 141.461,Z 887.023,A -85,B 0,C 180,E1 -19765.565,E2 -19765.565} C_VEL
LIN {X 0,Y 134.185,Z 889.621,A -85,B 0,C 180,E1 -19769.555,E2 -19769.555} C_VEL
LIN {X 0,Y 128.378,Z 891.824,A -85,B 0,C 180,E1 -19773.643,E2 -19773.643} C_VEL
LIN {X 0,Y 123.484,Z 893.877,A -85,B 0,C 180,E1 -19778.131,E2 -19778.131} C_VEL
LIN {X 0,Y 119.559,Z 895.814,A -85,B 0,C 180,E1 -19782.979,E2 -19782.979} C_VEL
LIN {X 0,Y 116.652,Z 897.674,A -85,B 0,C 180,E1 -19788.127,E2 -19788.127} C_VEL
LIN {X 0,Y 116.511,Z 897.913,A -85,B 0,C 180,E1 -19788.866,E2 -19788.866} C_VEL
LIN {X 0,Y 116.039,Z 908.168,A -85,B 0,C 180,E1 -19797.035,E2 -19797.035} C_VEL
LIN {X 0,Y 117.737,Z 917.684,A -85,B 0,C 180,E1 -19806.337,E2 -19806.337} C_VEL
LIN {X 0,Y 122.589,Z 925.862,A -85,B 0,C 180,E1 -19816.098,E2 -19816.098} C_VEL
LIN {X 0,Y 131.559,Z 932.461,A -85,B 0,C 180,E1 -19825.67,E2 -19825.67} C_VEL
LIN {X 0,Y 139.284,Z 935.582,A -85,B 0,C 180,E1 -19831.116,E2 -19831.116} C_VEL
LIN {X 0,Y 139.929,Z 936.168,A -85,B 0,C 180,E1 -19832.131,E2 -19832.131} C_VEL
LIN {X 0,Y 138.848,Z 937.107,A -85,B 0,C 180,E1 -19833.747,E2 -19833.747} C_VEL
LIN {X 0,Y 135.818,Z 938.092,A -85,B 0,C 180,E1 -19835.517,E2 -19835.517} C_VEL
LIN {X 0,Y 127.072,Z 940.116,A -85,B 0,C 180,E1 -19839.806,E2 -19839.806} C_VEL
LIN {X 0,Y 112.934,Z 944.72,A -85,B 0,C 180,E1 -19854.243,E2 -19854.243} C_VEL
LIN {X 0,Y 108.166,Z 946.892,A -85,B 0,C 180,E1 -19865.999,E2 -19865.999} C_VEL
LIN {X 0,Y 106.85,Z 950.763,A -85,B 0,C 180,E1 -19875.917,E2 -19875.917} C_VEL
LIN {X 0,Y 107.619,Z 952.743,A -85,B 0,C 180,E1 -19884.668,E2 -19884.668} C_VEL
LIN {X 0,Y 108.282,Z 953.168,A -85,B 0,C 180,E1 -19889.998,E2 -19889.998} C_VEL
LIN {X 0,Y 107.594,Z 952.726,A -85,B 0,C 180,E1 -19895.331,E2 -19895.331} C_VEL
LIN {X 0,Y 106.725,Z 950.721,A -85,B 0,C 180,E1 -19904.097,E2 -19904.097} C_VEL
LIN {X 0,Y 107.798,Z 946.791,A -85,B 0,C 180,E1 -19914.085,E2 -19914.085} C_VEL
LIN {X 0,Y 111.54,Z 941.08,A -85,B 0,C 180,E1 -19923.763,E2 -19923.763} C_VEL
LIN {X 0,Y 117.984,Z 933.51,A -85,B 0,C 180,E1 -19932.683,E2 -19932.683} C_VEL
LIN {X 0,Y 126.861,Z 923.917,A -85,B 0,C 180,E1 -19940.567,E2 -19940.567} C_VEL
LIN {X 0,Y 137.112,Z 912.677,A -85,B 0,C 180,E1 -19946.992,E2 -19946.992} C_VEL
LIN {X 0,Y 147.352,Z 900.732,A -85,B 0,C 180,E1 -19951.897,E2 -19951.897} C_VEL
LIN {X 0,Y 157.796,Z 887.486,A -85,B 0,C 180,E1 -19955.842,E2 -19955.842} C_VEL
LIN {X 0,Y 168.084,Z 872.79,A -85,B 0,C 180,E1 -19959.09,E2 -19959.09} C_VEL
LIN {X 0,Y 177.591,Z 857.418,A -85,B 0,C 180,E1 -19961.561,E2 -19961.561} C_VEL
LIN {X 0,Y 186.083,Z 841.26,A -85,B 0,C 180,E1 -19963.557,E2 -19963.557} C_VEL
LIN {X 0,Y 193.483,Z 824.519,A -85,B 0,C 180,E1 -19965.093,E2 -19965.093} C_VEL
LIN {X 0,Y 199.898,Z 806.515,A -85,B 0,C 180,E1 -19966.311,E2 -19966.311} C_VEL
LIN {X 0,Y 204.991,Z 787.659,A -85,B 0,C 180,E1 -19967.208,E2 -19967.208} C_VEL
LIN {X 0,Y 208.497,Z 768.703,A -85,B 0,C 180,E1 -19967.803,E2 -19967.803} C_VEL
LIN {X 0,Y 212.03,Z 737.114,A -85,B 0,C 180,E1 -19968.555,E2 -19968.555} C_VEL
LIN {X 0,Y 214.289,Z 716.605,A -85,B 0,C 180,E1 -19968.943,E2 -19968.943} C_VEL
LIN {X 0,Y 217.399,Z 690.669,A -85,B 0,C 180,E1 -19969.121,E2 -19969.121} C_VEL
LIN {X 0,Y 220.334,Z 668.167,A -85,B 0,C 180,E1 -19968.98,E2 -19968.98} C_VEL
LIN {X 0,Y 220.626,Z 665.959,A -85,B 0,C 180,E1 -19968.962,E2 -19968.962} C_VEL
LIN {X 0,Y 220.942,Z 645.734,A -85,B 0,C 180,E1 -19972.051,E2 -19972.051} C_VEL
LIN {X 0,Y 221.66,Z 635.777,A -85,B 0,C 180,E1 -19973.396,E2 -19973.396} C_VEL
LIN {X 0,Y 224.221,Z 623.761,A -85,B 0,C 180,E1 -19975.269,E2 -19975.269} C_VEL
LIN {X 0,Y 222.061,Z 618.693,A -85,B 0,C 180,E1 -19977.162,E2 -19977.162} C_VEL
LIN {X 0,Y 222.344,Z 612.366,A -85,B 0,C 180,E1 -19980.516,E2 -19980.516} C_VEL
LIN {X 0,Y 223.702,Z 605.087,A -85,B 0,C 180,E1 -19984.744,E2 -19984.744} C_VEL
LIN {X 0,Y 225.621,Z 599.838,A -85,B 0,C 180,E1 -19988.153,E2 -19988.153} C_VEL
LIN {X 0,Y 227.825,Z 595.788,A -85,B 0,C 180,E1 -19991.007,E2 -19991.007} C_VEL
LIN {X 0,Y 231.606,Z 590.851,A -85,B 0,C 180,E1 -19994.757,E2 -19994.757} C_VEL
LIN {X 0,Y 232.877,Z 589.789,A -85,B 0,C 180,E1 -19995.857,E2 -19995.857} C_VEL
LIN {X 0,Y 219.133,Z 722.145,A -85,B 0,C 180,E1 -19998.637,E2 -19998.637} C_VEL
LIN {X 0,Y 215.959,Z 753.933,A -85,B 0,C 180,E1 -19999.681,E2 -19999.681} C_VEL
LIN {X 0,Y 212.524,Z 772.732,A -85,B 0,C 180,E1 -20000.601,E2 -20000.601} C_VEL
LIN {X 0,Y 207.768,Z 790.414,A -85,B 0,C 180,E1 -20001.755,E2 -20001.755} C_VEL
LIN {X 0,Y 201.748,Z 807.265,A -85,B 0,C 180,E1 -20003.173,E2 -20003.173} C_VEL
LIN {X 0,Y 194.539,Z 823.38,A -85,B 0,C 180,E1 -20004.927,E2 -20004.927} C_VEL
LIN {X 0,Y 185.968,Z 839.119,A -85,B 0,C 180,E1 -20007.152,E2 -20007.152} C_VEL
LIN {X 0,Y 176.402,Z 853.823,A -85,B 0,C 180,E1 -20009.865,E2 -20009.865} C_VEL
LIN {X 0,Y 166.072,Z 867.371,A -85,B 0,C 180,E1 -20013.191,E2 -20013.191} C_VEL
LIN {X 0,Y 155.48,Z 879.404,A -85,B 0,C 180,E1 -20017.194,E2 -20017.194} C_VEL
LIN {X 0,Y 145.011,Z 889.845,A -85,B 0,C 180,E1 -20021.978,E2 -20021.978} C_VEL
LIN {X 0,Y 135.1,Z 898.656,A -85,B 0,C 180,E1 -20027.665,E2 -20027.665} C_VEL
LIN {X 0,Y 125.957,Z 906.041,A -85,B 0,C 180,E1 -20034.587,E2 -20034.587} C_VEL
LIN {X 0,Y 118.214,Z 911.793,A -85,B 0,C 180,E1 -20042.825,E2 -20042.825} C_VEL
LIN {X 0,Y 112.751,Z 915.667,A -85,B 0,C 180,E1 -20051.92,E2 -20051.92} C_VEL
LIN {X 0,Y 109.692,Z 917.829,A -85,B 0,C 180,E1 -20061.615,E2 -20061.615} C_VEL
LIN {X 0,Y 108.914,Z 918.403,A -85,B 0,C 180,E1 -20071.054,E2 -20071.054} C_VEL
LIN {X 0,Y 110.13,Z 917.561,A -85,B 0,C 180,E1 -20080.463,E2 -20080.463} C_VEL
LIN {X 0,Y 113.667,Z 915.07,A -85,B 0,C 180,E1 -20090.065,E2 -20090.065} C_VEL
LIN {X 0,Y 119.609,Z 910.824,A -85,B 0,C 180,E1 -20099.004,E2 -20099.004} C_VEL
LIN {X 0,Y 127.297,Z 905.055,A -85,B 0,C 180,E1 -20106.653,E2 -20106.653} C_VEL
LIN {X 0,Y 136.706,Z 897.395,A -85,B 0,C 180,E1 -20113.435,E2 -20113.435} C_VEL
LIN {X 0,Y 147.155,Z 887.963,A -85,B 0,C 180,E1 -20119.158,E2 -20119.158} C_VEL
LIN {X 0,Y 147.25,Z 887.789,A -85,B 0,C 180,E1 -20119.317,E2 -20119.317} C_VEL
LIN {X 0,Y 136.566,Z 891.253,A -85,B 0,C 180,E1 -20123.626,E2 -20123.626} C_VEL
LIN {X 0,Y 128.945,Z 893.809,A -85,B 0,C 180,E1 -20127.652,E2 -20127.652} C_VEL
LIN {X 0,Y 122.814,Z 895.988,A -85,B 0,C 180,E1 -20131.822,E2 -20131.822} C_VEL
LIN {X 0,Y 117.598,Z 898.029,A -85,B 0,C 180,E1 -20136.445,E2 -20136.445} C_VEL
LIN {X 0,Y 113.37,Z 899.968,A -85,B 0,C 180,E1 -20141.487,E2 -20141.487} C_VEL
LIN {X 0,Y 110.192,Z 901.836,A -85,B 0,C 180,E1 -20146.887,E2 -20146.887} C_VEL
LIN {X 0,Y 108.043,Z 903.792,A -85,B 0,C 180,E1 -20153.089,E2 -20153.089} C_VEL
LIN {X 0,Y 108.006,Z 904.577,A -85,B 0,C 180,E1 -20154.154,E2 -20154.154} C_VEL
LIN {X 0,Y 109.058,Z 915.084,A -85,B 0,C 180,E1 -20164.205,E2 -20164.205} C_VEL
LIN {X 0,Y 113.107,Z 923.834,A -85,B 0,C 180,E1 -20174.329,E2 -20174.329} C_VEL
LIN {X 0,Y 120.682,Z 930.935,A -85,B 0,C 180,E1 -20183.95,E2 -20183.95} C_VEL
LIN {X 0,Y 131.975,Z 936.41,A -85,B 0,C 180,E1 -20192.54,E2 -20192.54} C_VEL
LIN {X 0,Y 135.549,Z 937.591,A -85,B 0,C 180,E1 -20194.665,E2 -20194.665} C_VEL
LIN {X 0,Y 127.072,Z 940.116,A -85,B 0,C 180,E1 -20199.806,E2 -20199.806} C_VEL
LIN {X 0,Y 121.913,Z 941.181,A -85,B 0,C 180,E1 -20202.775,E2 -20202.775} C_VEL
LIN {X 0,Y 108.054,Z 942.389,A -85,B 0,C 180,E1 -20210.425,E2 -20210.425} C_VEL
LIN {X 0,Y 105.169,Z 942.843,A -85,B 0,C 180,E1 -20213.64,E2 -20213.64} C_VEL
LIN {X 0,Y 101.678,Z 944.194,A -85,B 0,C 180,E1 -20221.192,E2 -20221.192} C_VEL
LIN {X 0,Y 99.066,Z 948.739,A -85,B 0,C 180,E1 -20232.373,E2 -20232.373} C_VEL
LIN {X 0,Y 99.38,Z 951.16,A -85,B 0,C 180,E1 -20242.483,E2 -20242.483} C_VEL
LIN {X 0,Y 100.344,Z 951.884,A -85,B 0,C 180,E1 -20249.427,E2 -20249.427} C_VEL
LIN {X 0,Y 99.87,Z 951.63,A -85,B 0,C 180,E1 -20254.017,E2 -20254.017} C_VEL
LIN {X 0,Y 98.826,Z 950.028,A -85,B 0,C 180,E1 -20262.859,E2 -20262.859} C_VEL
LIN {X 0,Y 99.67,Z 946.474,A -85,B 0,C 180,E1 -20273.656,E2 -20273.656} C_VEL
LIN {X 0,Y 103.419,Z 941.152,A -85,B 0,C 180,E1 -20284.106,E2 -20284.106} C_VEL
LIN {X 0,Y 110.078,Z 933.988,A -85,B 0,C 180,E1 -20293.653,E2 -20293.653} C_VEL
LIN {X 0,Y 119.31,Z 924.838,A -85,B 0,C 180,E1 -20301.974,E2 -20301.974} C_VEL
LIN {X 0,Y 129.963,Z 914.141,A -85,B 0,C 180,E1 -20308.644,E2 -20308.644} C_VEL
LIN {X 0,Y 140.571,Z 902.743,A -85,B 0,C 180,E1 -20313.663,E2 -20313.663} C_VEL
LIN {X 0,Y 151.906,Z 889.444,A -85,B 0,C 180,E1 -20317.837,E2 -20317.837} C_VEL
LIN {X 0,Y 162.734,Z 875.1,A -85,B 0,C 180,E1 -20321.116,E2 -20321.116} C_VEL
LIN {X 0,Y 172.964,Z 859.683,A -85,B 0,C 180,E1 -20323.656,E2 -20323.656} C_VEL
LIN {X 0,Y 182.016,Z 843.651,A -85,B 0,C 180,E1 -20325.651,E2 -20325.651} C_VEL
LIN {X 0,Y 190.179,Z 826.434,A -85,B 0,C 180,E1 -20327.225,E2 -20327.225} C_VEL
LIN {X 0,Y 196.983,Z 808.702,A -85,B 0,C 180,E1 -20328.415,E2 -20328.415} C_VEL
LIN {X 0,Y 202.638,Z 789.504,A -85,B 0,C 180,E1 -20329.324,E2 -20329.324} C_VEL
LIN {X 0,Y 206.603,Z 769.933,A -85,B 0,C 180,E1 -20329.933,E2 -20329.933} C_VEL
LIN {X 0,Y 210.119,Z 740.205,A -85,B 0,C 180,E1 -20330.598,E2 -20330.598} C_VEL
LIN {X 0,Y 212.501,Z 718.761,A -85,B 0,C 180,E1 -20331.036,E2 -20331.036} C_VEL
LIN {X 0,Y 215.895,Z 690.637,A -85,B 0,C 180,E1 -20331.201,E2 -20331.201} C_VEL
LIN {X 0,Y 218.83,Z 667.632,A -85,B 0,C 180,E1 -20331.093,E2 -20331.093} C_VEL
LIN {X 0,Y 219.628,Z 647.262,A -85,B 0,C 180,E1 -20334.154,E2 -20334.154} C_VEL
LIN {X 0,Y 220.923,Z 628.916,A -85,B 0,C 180,E1 -20336.725,E2 -20336.725} C_VEL
LIN {X 0,Y 220.983,Z 625.108,A -85,B 0,C 180,E1 -20338.51,E2 -20338.51} C_VEL
LIN {X 0,Y 221.703,Z 617.987,A -85,B 0,C 180,E1 -20342.327,E2 -20342.327} C_VEL
LIN {X 0,Y 223.078,Z 612.28,A -85,B 0,C 180,E1 -20345.66,E2 -20345.66} C_VEL
LIN {X 0,Y 225.119,Z 607.208,A -85,B 0,C 180,E1 -20348.944,E2 -20348.944} C_VEL
LIN {X 0,Y 227.592,Z 603,A -85,B 0,C 180,E1 -20351.917,E2 -20351.917} C_VEL
LIN {X 0,Y 229.841,Z 600.076,A -85,B 0,C 180,E1 -20354.133,E2 -20354.133} C_VEL
LIN {X 0,Y 216.787,Z 722.694,A -85,B 0,C 180,E1 -20356.632,E2 -20356.632} C_VEL
LIN {X 0,Y 213.441,Z 755.029,A -85,B 0,C 180,E1 -20357.674,E2 -20357.674} C_VEL
LIN {X 0,Y 209.901,Z 773.841,A -85,B 0,C 180,E1 -20358.573,E2 -20358.573} C_VEL
LIN {X 0,Y 204.97,Z 791.654,A -85,B 0,C 180,E1 -20359.702,E2 -20359.702} C_VEL
LIN {X 0,Y 198.771,Z 808.512,A -85,B 0,C 180,E1 -20361.079,E2 -20361.079} C_VEL
LIN {X 0,Y 191.43,Z 824.466,A -85,B 0,C 180,E1 -20362.761,E2 -20362.761} C_VEL
LIN {X 0,Y 182.899,Z 839.735,A -85,B 0,C 180,E1 -20364.843,E2 -20364.843} C_VEL
LIN {X 0,Y 173.383,Z 854.019,A -85,B 0,C 180,E1 -20367.369,E2 -20367.369} C_VEL
LIN {X 0,Y 163.384,Z 866.864,A -85,B 0,C 180,E1 -20370.361,E2 -20370.361} C_VEL
LIN {X 0,Y 153.059,Z 878.378,A -85,B 0,C 180,E1 -20373.941,E2 -20373.941} C_VEL
LIN {X 0,Y 141.945,Z 889.197,A -85,B 0,C 180,E1 -20378.568,E2 -20378.568} C_VEL
LIN {X 0,Y 131.131,Z 898.47,A -85,B 0,C 180,E1 -20384.216,E2 -20384.216} C_VEL
LIN {X 0,Y 121.089,Z 906.174,A -85,B 0,C 180,E1 -20391.132,E2 -20391.132} C_VEL
LIN {X 0,Y 112.793,Z 911.98,A -85,B 0,C 180,E1 -20399.061,E2 -20399.061} C_VEL
LIN {X 0,Y 106.297,Z 916.257,A -85,B 0,C 180,E1 -20408.48,E2 -20408.48} C_VEL
LIN {X 0,Y 102.381,Z 918.782,A -85,B 0,C 180,E1 -20418.738,E2 -20418.738} C_VEL
LIN {X 0,Y 101.01,Z 919.679,A -85,B 0,C 180,E1 -20429.434,E2 -20429.434} C_VEL
LIN {X 0,Y 102.104,Z 918.999,A -85,B 0,C 180,E1 -20440.154,E2 -20440.154} C_VEL
LIN {X 0,Y 105.898,Z 916.594,A -85,B 0,C 180,E1 -20450.812,E2 -20450.812} C_VEL
LIN {X 0,Y 112.343,Z 912.37,A -85,B 0,C 180,E1 -20460.486,E2 -20460.486} C_VEL
LIN {X 0,Y 120.523,Z 906.699,A -85,B 0,C 180,E1 -20468.479,E2 -20468.479} C_VEL
LIN {X 0,Y 129.875,Z 899.627,A -85,B 0,C 180,E1 -20475.096,E2 -20475.096} C_VEL
LIN {X 0,Y 137.044,Z 893.644,A -85,B 0,C 180,E1 -20479.204,E2 -20479.204} C_VEL
LIN {X 0,Y 123.732,Z 897.736,A -85,B 0,C 180,E1 -20485.55,E2 -20485.55} C_VEL
LIN {X 0,Y 117.253,Z 899.888,A -85,B 0,C 180,E1 -20489.792,E2 -20489.792} C_VEL
LIN {X 0,Y 111.292,Z 902.056,A -85,B 0,C 180,E1 -20495.021,E2 -20495.021} C_VEL
LIN {X 0,Y 106.829,Z 903.98,A -85,B 0,C 180,E1 -20500.308,E2 -20500.308} C_VEL
LIN {X 0,Y 103.459,Z 905.84,A -85,B 0,C 180,E1 -20506.017,E2 -20506.017} C_VEL
LIN {X 0,Y 101.226,Z 907.678,A -85,B 0,C 180,E1 -20512.05,E2 -20512.05} C_VEL
LIN {X 0,Y 100.165,Z 909.659,A -85,B 0,C 180,E1 -20518.854,E2 -20518.854} C_VEL
LIN {X 0,Y 100.285,Z 910.324,A -85,B 0,C 180,E1 -20519.998,E2 -20519.998} C_VEL
LIN {X 0,Y 103.251,Z 920.376,A -85,B 0,C 180,E1 -20531.166,E2 -20531.166} C_VEL
LIN {X 0,Y 109.947,Z 928.661,A -85,B 0,C 180,E1 -20541.89,E2 -20541.89} C_VEL
LIN {X 0,Y 120.073,Z 935.028,A -85,B 0,C 180,E1 -20551.081,E2 -20551.081} C_VEL
LIN {X 0,Y 125.44,Z 937.319,A -85,B 0,C 180,E1 -20554.685,E2 -20554.685} C_VEL
LIN {X 0,Y 107.913,Z 942.029,A -85,B 0,C 180,E1 -20569.563,E2 -20569.563} C_VEL
LIN {X 0,Y 105.169,Z 942.843,A -85,B 0,C 180,E1 -20573.64,E2 -20573.64} C_VEL
LIN {X 0,Y 102.07,Z 943.679,A -85,B 0,C 180,E1 -20577.546,E2 -20577.546} C_VEL
LIN {X 0,Y 91.96,Z 947.052,A -85,B 0,C 180,E1 -20589.23,E2 -20589.23} C_VEL
LIN {X 0,Y 91.095,Z 947.958,A -85,B 0,C 180,E1 -20592.635,E2 -20592.635} C_VEL
LIN {X 0,Y 91.594,Z 950.167,A -85,B 0,C 180,E1 -20603.731,E2 -20603.731} C_VEL
LIN {X 0,Y 92.471,Z 950.64,A -85,B 0,C 180,E1 -20609.998,E2 -20609.998} C_VEL
LIN {X 0,Y 91.47,Z 950.048,A -85,B 0,C 180,E1 -20616.904,E2 -20616.904} C_VEL
LIN {X 0,Y 90.919,Z 947.759,A -85,B 0,C 180,E1 -20627.932,E2 -20627.932} C_VEL
LIN {X 0,Y 93.321,Z 943.495,A -85,B 0,C 180,E1 -20639.794,E2 -20639.794} C_VEL
LIN {X 0,Y 99.174,Z 937.27,A -85,B 0,C 180,E1 -20650.942,E2 -20650.942} C_VEL
LIN {X 0,Y 107.807,Z 929.345,A -85,B 0,C 180,E1 -20660.332,E2 -20660.332} C_VEL
LIN {X 0,Y 118.158,Z 919.969,A -85,B 0,C 180,E1 -20667.799,E2 -20667.799} C_VEL
LIN {X 0,Y 129.412,Z 909.22,A -85,B 0,C 180,E1 -20673.665,E2 -20673.665} C_VEL
LIN {X 0,Y 141.458,Z 896.626,A -85,B 0,C 180,E1 -20678.437,E2 -20678.437} C_VEL
LIN {X 0,Y 153.65,Z 882.355,A -85,B 0,C 180,E1 -20682.192,E2 -20682.192} C_VEL
LIN {X 0,Y 164.588,Z 867.659,A -85,B 0,C 180,E1 -20684.994,E2 -20684.994} C_VEL
LIN {X 0,Y 174.834,Z 851.747,A -85,B 0,C 180,E1 -20687.177,E2 -20687.177} C_VEL
LIN {X 0,Y 183.817,Z 835.252,A -85,B 0,C 180,E1 -20688.825,E2 -20688.825} C_VEL
LIN {X 0,Y 191.277,Z 818.636,A -85,B 0,C 180,E1 -20690.086,E2 -20690.086} C_VEL
LIN {X 0,Y 197.617,Z 801.015,A -85,B 0,C 180,E1 -20691.067,E2 -20691.067} C_VEL
LIN {X 0,Y 202.635,Z 782.501,A -85,B 0,C 180,E1 -20691.776,E2 -20691.776} C_VEL
LIN {X 0,Y 206.033,Z 763.99,A -85,B 0,C 180,E1 -20692.228,E2 -20692.228} C_VEL
LIN {X 0,Y 211.079,Z 720.276,A -85,B 0,C 180,E1 -20693.162,E2 -20693.162} C_VEL
LIN {X 0,Y 214.668,Z 690.694,A -85,B 0,C 180,E1 -20693.307,E2 -20693.307} C_VEL
LIN {X 0,Y 217.335,Z 669.533,A -85,B 0,C 180,E1 -20693.214,E2 -20693.214} C_VEL
LIN {X 0,Y 218.609,Z 648.863,A -85,B 0,C 180,E1 -20696.264,E2 -20696.264} C_VEL
LIN {X 0,Y 219.863,Z 634.516,A -85,B 0,C 180,E1 -20698.307,E2 -20698.307} C_VEL
LIN {X 0,Y 220.053,Z 631.247,A -85,B 0,C 180,E1 -20700.001,E2 -20700.001} C_VEL
LIN {X 0,Y 220.934,Z 625.148,A -85,B 0,C 180,E1 -20703.244,E2 -20703.244} C_VEL
LIN {X 0,Y 222.512,Z 619.461,A -85,B 0,C 180,E1 -20706.58,E2 -20706.58} C_VEL
LIN {X 0,Y 224.857,Z 614.228,A -85,B 0,C 180,E1 -20709.987,E2 -20709.987} C_VEL
LIN {X 0,Y 226.967,Z 610.823,A -85,B 0,C 180,E1 -20712.37,E2 -20712.37} C_VEL
LIN {X 0,Y 214.706,Z 723.311,A -85,B 0,C 180,E1 -20714.586,E2 -20714.586} C_VEL
LIN {X 0,Y 211.159,Z 756.312,A -85,B 0,C 180,E1 -20715.631,E2 -20715.631} C_VEL
LIN {X 0,Y 207.49,Z 775.175,A -85,B 0,C 180,E1 -20716.508,E2 -20716.508} C_VEL
LIN {X 0,Y 202.442,Z 792.895,A -85,B 0,C 180,E1 -20717.596,E2 -20717.596} C_VEL
LIN {X 0,Y 196.068,Z 809.76,A -85,B 0,C 180,E1 -20718.923,E2 -20718.923} C_VEL
LIN {X 0,Y 188.471,Z 825.797,A -85,B 0,C 180,E1 -20720.555,E2 -20720.555} C_VEL
LIN {X 0,Y 179.537,Z 841.276,A -85,B 0,C 180,E1 -20722.599,E2 -20722.599} C_VEL
LIN {X 0,Y 169.894,Z 855.278,A -85,B 0,C 180,E1 -20725,E2 -20725} C_VEL
LIN {X 0,Y 159.532,Z 868.126,A -85,B 0,C 180,E1 -20727.909,E2 -20727.909} C_VEL
LIN {X 0,Y 148.785,Z 879.642,A -85,B 0,C 180,E1 -20731.412,E2 -20731.412} C_VEL
LIN {X 0,Y 137.147,Z 890.462,A -85,B 0,C 180,E1 -20735.981,E2 -20735.981} C_VEL
LIN {X 0,Y 125.734,Z 899.736,A -85,B 0,C 180,E1 -20741.627,E2 -20741.627} C_VEL
LIN {X 0,Y 115.025,Z 907.441,A -85,B 0,C 180,E1 -20748.654,E2 -20748.654} C_VEL
LIN {X 0,Y 106.074,Z 913.248,A -85,B 0,C 180,E1 -20756.86,E2 -20756.86} C_VEL
LIN {X 0,Y 98.973,Z 917.524,A -85,B 0,C 180,E1 -20766.799,E2 -20766.799} C_VEL
LIN {X 0,Y 94.639,Z 920.047,A -85,B 0,C 180,E1 -20777.803,E2 -20777.803} C_VEL
LIN {X 0,Y 93.111,Z 920.943,A -85,B 0,C 180,E1 -20789.386,E2 -20789.386} C_VEL
LIN {X 0,Y 94.332,Z 920.263,A -85,B 0,C 180,E1 -20801.001,E2 -20801.001} C_VEL
LIN {X 0,Y 98.356,Z 917.968,A -85,B 0,C 180,E1 -20812.096,E2 -20812.096} C_VEL
LIN {X 0,Y 105.249,Z 913.86,A -85,B 0,C 180,E1 -20822.272,E2 -20822.272} C_VEL
LIN {X 0,Y 114.423,Z 907.964,A -85,B 0,C 180,E1 -20830.95,E2 -20830.95} C_VEL
LIN {X 0,Y 124.407,Z 900.89,A -85,B 0,C 180,E1 -20837.683,E2 -20837.683} C_VEL
LIN {X 0,Y 126.941,Z 898.935,A -85,B 0,C 180,E1 -20839.173,E2 -20839.173} C_VEL
LIN {X 0,Y 113.407,Z 903.019,A -85,B 0,C 180,E1 -20846.257,E2 -20846.257} C_VEL
LIN {X 0,Y 100.521,Z 907.592,A -85,B 0,C 180,E1 -20858.404,E2 -20858.404} C_VEL
LIN {X 0,Y 94.221,Z 911.407,A -85,B 0,C 180,E1 -20871.454,E2 -20871.454} C_VEL
LIN {X 0,Y 93.555,Z 915.56,A -85,B 0,C 180,E1 -20886.75,E2 -20886.75} C_VEL
LIN {X 0,Y 99.022,Z 925.226,A -85,B 0,C 180,E1 -20898.85,E2 -20898.85} C_VEL
LIN {X 0,Y 108.306,Z 932.795,A -85,B 0,C 180,E1 -20909.292,E2 -20909.292} C_VEL
LIN {X 0,Y 115.519,Z 936.544,A -85,B 0,C 180,E1 -20914.686,E2 -20914.686} C_VEL
LIN {X 0,Y 98.988,Z 940.357,A -85,B 0,C 180,E1 -20930.477,E2 -20930.477} C_VEL
LIN {X 0,Y 96.313,Z 941.051,A -85,B 0,C 180,E1 -20935.18,E2 -20935.18} C_VEL
LIN {X 0,Y 91.855,Z 946.201,A -85,B 0,C 180,E1 -20946.927,E2 -20946.927} C_VEL
LIN {X 0,Y 91.095,Z 947.958,A -85,B 0,C 180,E1 -20952.635,E2 -20952.635} C_VEL
LIN {X 0,Y 90.148,Z 949.003,A -85,B 0,C 180,E1 -20957.494,E2 -20957.494} C_VEL
LIN {X 0,Y 87.851,Z 949.57,A -85,B 0,C 180,E1 -20963.446,E2 -20963.446} C_VEL
LIN {X 0,Y 83.879,Z 949.078,A -85,B 0,C 180,E1 -20974.644,E2 -20974.644} C_VEL
LIN {X 0,Y 83.673,Z 948.975,A -85,B 0,C 180,E1 -20975.814,E2 -20975.814} C_VEL
LIN {X 0,Y 82.966,Z 946.867,A -85,B 0,C 180,E1 -20987.819,E2 -20987.819} C_VEL
LIN {X 0,Y 85.553,Z 942.786,A -85,B 0,C 180,E1 -21000.944,E2 -21000.944} C_VEL
LIN {X 0,Y 91.638,Z 937.043,A -85,B 0,C 180,E1 -21012.567,E2 -21012.567} C_VEL
LIN {X 0,Y 100.828,Z 929.457,A -85,B 0,C 180,E1 -21022.494,E2 -21022.494} C_VEL
LIN {X 0,Y 112.461,Z 919.86,A -85,B 0,C 180,E1 -21030.606,E2 -21030.606} C_VEL
LIN {X 0,Y 125.103,Z 908.62,A -85,B 0,C 180,E1 -21036.794,E2 -21036.794} C_VEL
LIN {X 0,Y 137.552,Z 896.382,A -85,B 0,C 180,E1 -21041.348,E2 -21041.348} C_VEL
LIN {X 0,Y 149.705,Z 882.939,A -85,B 0,C 180,E1 -21044.813,E2 -21044.813} C_VEL
LIN {X 0,Y 161.269,Z 868.221,A -85,B 0,C 180,E1 -21047.547,E2 -21047.547} C_VEL
LIN {X 0,Y 171.817,Z 852.655,A -85,B 0,C 180,E1 -21049.608,E2 -21049.608} C_VEL
LIN {X 0,Y 181.121,Z 836.436,A -85,B 0,C 180,E1 -21051.165,E2 -21051.165} C_VEL
LIN {X 0,Y 188.96,Z 819.923,A -85,B 0,C 180,E1 -21052.372,E2 -21052.372} C_VEL
LIN {X 0,Y 195.798,Z 801.952,A -85,B 0,C 180,E1 -21053.323,E2 -21053.323} C_VEL
LIN {X 0,Y 201.217,Z 783.034,A -85,B 0,C 180,E1 -21054.005,E2 -21054.005} C_VEL
LIN {X 0,Y 204.949,Z 763.815,A -85,B 0,C 180,E1 -21054.439,E2 -21054.439} C_VEL
LIN {X 0,Y 210.075,Z 720.762,A -85,B 0,C 180,E1 -21055.32,E2 -21055.32} C_VEL
LIN {X 0,Y 213.744,Z 690.658,A -85,B 0,C 180,E1 -21055.434,E2 -21055.434} C_VEL
LIN {X 0,Y 216.139,Z 671.515,A -85,B 0,C 180,E1 -21055.34,E2 -21055.34} C_VEL
LIN {X 0,Y 217.855,Z 650.805,A -85,B 0,C 180,E1 -21058.341,E2 -21058.341} C_VEL
LIN {X 0,Y 218.978,Z 640.044,A -85,B 0,C 180,E1 -21059.929,E2 -21059.929} C_VEL
LIN {X 0,Y 220.302,Z 631.993,A -85,B 0,C 180,E1 -21064.361,E2 -21064.361} C_VEL
LIN {X 0,Y 222.005,Z 626.635,A -85,B 0,C 180,E1 -21067.506,E2 -21067.506} C_VEL
LIN {X 0,Y 224.275,Z 621.895,A -85,B 0,C 180,E1 -21070.568,E2 -21070.568} C_VEL
LIN {X 0,Y 212.895,Z 724.009,A -85,B 0,C 180,E1 -21072.506,E2 -21072.506} C_VEL
LIN {X 0,Y 209.17,Z 757.485,A -85,B 0,C 180,E1 -21073.54,E2 -21073.54} C_VEL
LIN {X 0,Y 205.383,Z 776.401,A -85,B 0,C 180,E1 -21074.391,E2 -21074.391} C_VEL
LIN {X 0,Y 200.194,Z 794.135,A -85,B 0,C 180,E1 -21075.438,E2 -21075.438} C_VEL
LIN {X 0,Y 193.531,Z 811.27,A -85,B 0,C 180,E1 -21076.734,E2 -21076.734} C_VEL
LIN {X 0,Y 185.412,Z 827.83,A -85,B 0,C 180,E1 -21078.361,E2 -21078.361} C_VEL
LIN {X 0,Y 175.988,Z 843.529,A -85,B 0,C 180,E1 -21080.378,E2 -21080.378} C_VEL
LIN {X 0,Y 165.454,Z 858.132,A -85,B 0,C 180,E1 -21082.845,E2 -21082.845} C_VEL
LIN {X 0,Y 154.364,Z 871.157,A -85,B 0,C 180,E1 -21085.799,E2 -21085.799} C_VEL
LIN {X 0,Y 142.484,Z 883.104,A -85,B 0,C 180,E1 -21089.526,E2 -21089.526} C_VEL
LIN {X 0,Y 130.453,Z 893.533,A -85,B 0,C 180,E1 -21094.132,E2 -21094.132} C_VEL
LIN {X 0,Y 118.613,Z 902.456,A -85,B 0,C 180,E1 -21099.908,E2 -21099.908} C_VEL
LIN {X 0,Y 107.465,Z 909.843,A -85,B 0,C 180,E1 -21107.221,E2 -21107.221} C_VEL
LIN {X 0,Y 97.674,Z 915.595,A -85,B 0,C 180,E1 -21116.444,E2 -21116.444} C_VEL
LIN {X 0,Y 90.476,Z 919.466,A -85,B 0,C 180,E1 -21127.247,E2 -21127.247} C_VEL
LIN {X 0,Y 86.301,Z 921.621,A -85,B 0,C 180,E1 -21139.319,E2 -21139.319} C_VEL
LIN {X 0,Y 85.22,Z 922.193,A -85,B 0,C 180,E1 -21151.347,E2 -21151.347} C_VEL
LIN {X 0,Y 86.907,Z 921.354,A -85,B 0,C 180,E1 -21163.305,E2 -21163.305} C_VEL
LIN {X 0,Y 91.787,Z 918.826,A -85,B 0,C 180,E1 -21175.288,E2 -21175.288} C_VEL
LIN {X 0,Y 99.487,Z 914.621,A -85,B 0,C 180,E1 -21185.658,E2 -21185.658} C_VEL
LIN {X 0,Y 109.145,Z 908.851,A -85,B 0,C 180,E1 -21194.127,E2 -21194.127} C_VEL
LIN {X 0,Y 116.584,Z 903.98,A -85,B 0,C 180,E1 -21199.002,E2 -21199.002} C_VEL
LIN {X 0,Y 99.942,Z 908.867,A -85,B 0,C 180,E1 -21209.983,E2 -21209.983} C_VEL
LIN {X 0,Y 87.34,Z 914.597,A -85,B 0,C 180,E1 -21229.444,E2 -21229.444} C_VEL
LIN {X 0,Y 88.744,Z 921.35,A -85,B 0,C 180,E1 -21255.686,E2 -21255.686} C_VEL
LIN {X 0,Y 97.688,Z 930.452,A -85,B 0,C 180,E1 -21268.086,E2 -21268.086} C_VEL
LIN {X 0,Y 105.626,Z 935.244,A -85,B 0,C 180,E1 -21274.771,E2 -21274.771} C_VEL
LIN {X 0,Y 91.667,Z 938.023,A -85,B 0,C 180,E1 -21289.119,E2 -21289.119} C_VEL
LIN {X 0,Y 85.156,Z 943.834,A -85,B 0,C 180,E1 -21301.713,E2 -21301.713} C_VEL
LIN {X 0,Y 83.056,Z 947.451,A -85,B 0,C 180,E1 -21314.64,E2 -21314.64} C_VEL
LIN {X 0,Y 83.975,Z 949.12,A -85,B 0,C 180,E1 -21325.901,E2 -21325.901} C_VEL
LIN {X 0,Y 84.509,Z 949.347,A -85,B 0,C 180,E1 -21330.676,E2 -21330.676} C_VEL
LIN {X 0,Y 83.673,Z 948.975,A -85,B 0,C 180,E1 -21335.814,E2 -21335.814} C_VEL
LIN {X 0,Y 82.248,Z 948.303,A -85,B 0,C 180,E1 -21340.663,E2 -21340.663} C_VEL
LIN {X 0,Y 78.872,Z 946.507,A -85,B 0,C 180,E1 -21348.149,E2 -21348.149} C_VEL
LIN {X 0,Y 76.711,Z 943.844,A -85,B 0,C 180,E1 -21356.948,E2 -21356.948} C_VEL
LIN {X 0,Y 77.248,Z 942.651,A -85,B 0,C 180,E1 -21360.581,E2 -21360.581} C_VEL
LIN {X 0,Y 83.734,Z 937.117,A -85,B 0,C 180,E1 -21373.831,E2 -21373.831} C_VEL
LIN {X 0,Y 93.963,Z 929.516,A -85,B 0,C 180,E1 -21384.93,E2 -21384.93} C_VEL
LIN {X 0,Y 106.32,Z 920.214,A -85,B 0,C 180,E1 -21393.301,E2 -21393.301} C_VEL
LIN {X 0,Y 119.311,Z 909.606,A -85,B 0,C 180,E1 -21399.394,E2 -21399.394} C_VEL
LIN {X 0,Y 132.179,Z 897.882,A -85,B 0,C 180,E1 -21403.876,E2 -21403.876} C_VEL
LIN {X 0,Y 144.655,Z 885.049,A -85,B 0,C 180,E1 -21407.223,E2 -21407.223} C_VEL
LIN {X 0,Y 156.889,Z 870.528,A -85,B 0,C 180,E1 -21409.937,E2 -21409.937} C_VEL
LIN {X 0,Y 168.129,Z 855.027,A -85,B 0,C 180,E1 -21411.953,E2 -21411.953} C_VEL
LIN {X 0,Y 177.523,Z 839.707,A -85,B 0,C 180,E1 -21413.413,E2 -21413.413} C_VEL
LIN {X 0,Y 185.803,Z 823.561,A -85,B 0,C 180,E1 -21414.577,E2 -21414.577} C_VEL
LIN {X 0,Y 193.069,Z 806.141,A -85,B 0,C 180,E1 -21415.488,E2 -21415.488} C_VEL
LIN {X 0,Y 199.101,Z 787.345,A -85,B 0,C 180,E1 -21416.17,E2 -21416.17} C_VEL
LIN {X 0,Y 203.452,Z 768.049,A -85,B 0,C 180,E1 -21416.62,E2 -21416.62} C_VEL
LIN {X 0,Y 207.592,Z 736.146,A -85,B 0,C 180,E1 -21417.269,E2 -21417.269} C_VEL
LIN {X 0,Y 210.966,Z 708.113,A -85,B 0,C 180,E1 -21417.583,E2 -21417.583} C_VEL
LIN {X 0,Y 213.921,Z 684.228,A -85,B 0,C 180,E1 -21417.499,E2 -21417.499} C_VEL
LIN {X 0,Y 215.245,Z 673.484,A -85,B 0,C 180,E1 -21417.481,E2 -21417.481} C_VEL
LIN {X 0,Y 217.379,Z 652.846,A -85,B 0,C 180,E1 -21420.413,E2 -21420.413} C_VEL
LIN {X 0,Y 218.19,Z 646.195,A -85,B 0,C 180,E1 -21421.445,E2 -21421.445} C_VEL
LIN {X 0,Y 219.692,Z 639.033,A -85,B 0,C 180,E1 -21425.354,E2 -21425.354} C_VEL
LIN {X 0,Y 221.557,Z 633.803,A -85,B 0,C 180,E1 -21428.435,E2 -21428.435} C_VEL
LIN {X 0,Y 221.744,Z 633.528,A -85,B 0,C 180,E1 -21428.732,E2 -21428.732} C_VEL
LIN {X 0,Y 211.345,Z 724.91,A -85,B 0,C 180,E1 -21430.398,E2 -21430.398} C_VEL
LIN {X 0,Y 207.459,Z 758.686,A -85,B 0,C 180,E1 -21431.414,E2 -21431.414} C_VEL
LIN {X 0,Y 203.561,Z 777.629,A -85,B 0,C 180,E1 -21432.234,E2 -21432.234} C_VEL
LIN {X 0,Y 198.236,Z 795.375,A -85,B 0,C 180,E1 -21433.236,E2 -21433.236} C_VEL
LIN {X 0,Y 191.378,Z 812.577,A -85,B 0,C 180,E1 -21434.473,E2 -21434.473} C_VEL
LIN {X 0,Y 183.076,Z 829.082,A -85,B 0,C 180,E1 -21436.013,E2 -21436.013} C_VEL
LIN {X 0,Y 173.394,Z 844.785,A -85,B 0,C 180,E1 -21437.929,E2 -21437.929} C_VEL
LIN {X 0,Y 162.548,Z 859.391,A -85,B 0,C 180,E1 -21440.276,E2 -21440.276} C_VEL
LIN {X 0,Y 151.089,Z 872.418,A -85,B 0,C 180,E1 -21443.097,E2 -21443.097} C_VEL
LIN {X 0,Y 138.754,Z 884.368,A -85,B 0,C 180,E1 -21446.681,E2 -21446.681} C_VEL
LIN {X 0,Y 126.18,Z 894.798,A -85,B 0,C 180,E1 -21451.154,E2 -21451.154} C_VEL
LIN {X 0,Y 113.692,Z 903.723,A -85,B 0,C 180,E1 -21456.844,E2 -21456.844} C_VEL
LIN {X 0,Y 101.617,Z 911.214,A -85,B 0,C 180,E1 -21464.317,E2 -21464.317} C_VEL
LIN {X 0,Y 91.177,Z 916.862,A -85,B 0,C 180,E1 -21473.691,E2 -21473.691} C_VEL
LIN {X 0,Y 83.232,Z 920.732,A -85,B 0,C 180,E1 -21485.139,E2 -21485.139} C_VEL
LIN {X 0,Y 78.548,Z 922.885,A -85,B 0,C 180,E1 -21498.251,E2 -21498.251} C_VEL
LIN {X 0,Y 77.322,Z 923.456,A -85,B 0,C 180,E1 -21511.484,E2 -21511.484} C_VEL
LIN {X 0,Y 79.232,Z 922.618,A -85,B 0,C 180,E1 -21524.621,E2 -21524.621} C_VEL
LIN {X 0,Y 84.615,Z 920.131,A -85,B 0,C 180,E1 -21537.444,E2 -21537.444} C_VEL
LIN {X 0,Y 93.162,Z 915.886,A -85,B 0,C 180,E1 -21548.5,E2 -21548.5} C_VEL
LIN {X 0,Y 103.602,Z 910.116,A -85,B 0,C 180,E1 -21557.181,E2 -21557.181} C_VEL
LIN {X 0,Y 106.187,Z 908.57,A -85,B 0,C 180,E1 -21558.99,E2 -21558.99} C_VEL
LIN {X 0,Y 88.406,Z 913.824,A -85,B 0,C 180,E1 -21573.1,E2 -21573.1} C_VEL
LIN {X 0,Y 86.211,Z 926.603,A -85,B 0,C 180,E1 -21625.409,E2 -21625.409} C_VEL
LIN {X 0,Y 95.782,Z 933.545,A -85,B 0,C 180,E1 -21635.037,E2 -21635.037} C_VEL
LIN {X 0,Y 88.153,Z 934.893,A -85,B 0,C 180,E1 -21642.5,E2 -21642.5} C_VEL
LIN {X 0,Y 79.665,Z 941.082,A -85,B 0,C 180,E1 -21654.734,E2 -21654.734} C_VEL
LIN {X 0,Y 75.509,Z 945.355,A -85,B 0,C 180,E1 -21669.049,E2 -21669.049} C_VEL
LIN {X 0,Y 75.628,Z 947.665,A -85,B 0,C 180,E1 -21683.164,E2 -21683.164} C_VEL
LIN {X 0,Y 76.646,Z 948.109,A -85,B 0,C 180,E1 -21689.998,E2 -21689.998} C_VEL
LIN {X 0,Y 75.191,Z 947.194,A -85,B 0,C 180,E1 -21700.27,E2 -21700.27} C_VEL
LIN {X 0,Y 75.736,Z 944.441,A -85,B 0,C 180,E1 -21714.372,E2 -21714.372} C_VEL
LIN {X 0,Y 77.248,Z 942.651,A -85,B 0,C 180,E1 -21720.581,E2 -21720.581} C_VEL
LIN {X 0,Y 78.293,Z 940.732,A -85,B 0,C 180,E1 -21726.062,E2 -21726.062} C_VEL
LIN {X 0,Y 80.785,Z 934.323,A -85,B 0,C 180,E1 -21740.615,E2 -21740.615} C_VEL
LIN {X 0,Y 83.613,Z 931.968,A -85,B 0,C 180,E1 -21744.505,E2 -21744.505} C_VEL
LIN {X 0,Y 95.874,Z 923.753,A -85,B 0,C 180,E1 -21753.748,E2 -21753.748} C_VEL
LIN {X 0,Y 109.28,Z 914.038,A -85,B 0,C 180,E1 -21760.454,E2 -21760.454} C_VEL
LIN {X 0,Y 123.011,Z 902.869,A -85,B 0,C 180,E1 -21765.407,E2 -21765.407} C_VEL
LIN {X 0,Y 136.471,Z 890.439,A -85,B 0,C 180,E1 -21769.033,E2 -21769.033} C_VEL
LIN {X 0,Y 149.488,Z 876.547,A -85,B 0,C 180,E1 -21771.844,E2 -21771.844} C_VEL
LIN {X 0,Y 161.395,Z 861.809,A -85,B 0,C 180,E1 -21773.878,E2 -21773.878} C_VEL
LIN {X 0,Y 172.011,Z 846.29,A -85,B 0,C 180,E1 -21775.469,E2 -21775.469} C_VEL
LIN {X 0,Y 181.774,Z 829.229,A -85,B 0,C 180,E1 -21776.713,E2 -21776.713} C_VEL
LIN {X 0,Y 190.131,Z 811.229,A -85,B 0,C 180,E1 -21777.649,E2 -21777.649} C_VEL
LIN {X 0,Y 196.99,Z 792.1,A -85,B 0,C 180,E1 -21778.335,E2 -21778.335} C_VEL
LIN {X 0,Y 201.951,Z 772.846,A -85,B 0,C 180,E1 -21778.79,E2 -21778.79} C_VEL
LIN {X 0,Y 204.977,Z 754.702,A -85,B 0,C 180,E1 -21779.12,E2 -21779.12} C_VEL
LIN {X 0,Y 209.159,Z 720.202,A -85,B 0,C 180,E1 -21779.69,E2 -21779.69} C_VEL
LIN {X 0,Y 212.842,Z 690.16,A -85,B 0,C 180,E1 -21779.724,E2 -21779.724} C_VEL
LIN {X 0,Y 214.68,Z 675.223,A -85,B 0,C 180,E1 -21779.667,E2 -21779.667} C_VEL
LIN {X 0,Y 217.537,Z 652.418,A -85,B 0,C 180,E1 -21782.899,E2 -21782.899} C_VEL
LIN {X 0,Y 219.076,Z 646.283,A -85,B 0,C 180,E1 -21786.224,E2 -21786.224} C_VEL
LIN {X 0,Y 219.419,Z 645.398,A -85,B 0,C 180,E1 -21786.856,E2 -21786.856} C_VEL
LIN {X 0,Y 210.015,Z 726.446,A -85,B 0,C 180,E1 -21788.277,E2 -21788.277} C_VEL
LIN {X 0,Y 206.008,Z 760.059,A -85,B 0,C 180,E1 -21789.261,E2 -21789.261} C_VEL
LIN {X 0,Y 202.004,Z 778.962,A -85,B 0,C 180,E1 -21790.047,E2 -21790.047} C_VEL
LIN {X 0,Y 196.577,Z 796.616,A -85,B 0,C 180,E1 -21790.992,E2 -21790.992} C_VEL
LIN {X 0,Y 189.71,Z 813.503,A -85,B 0,C 180,E1 -21792.135,E2 -21792.135} C_VEL
LIN {X 0,Y 181.511,Z 829.554,A -85,B 0,C 180,E1 -21793.531,E2 -21793.531} C_VEL
LIN {X 0,Y 172.027,Z 844.759,A -85,B 0,C 180,E1 -21795.244,E2 -21795.244} C_VEL
LIN {X 0,Y 161.309,Z 859.055,A -85,B 0,C 180,E1 -21797.343,E2 -21797.343} C_VEL
LIN {X 0,Y 149.674,Z 872.14,A -85,B 0,C 180,E1 -21799.92,E2 -21799.92} C_VEL
LIN {X 0,Y 137.063,Z 884.166,A -85,B 0,C 180,E1 -21803.2,E2 -21803.2} C_VEL
LIN {X 0,Y 123.875,Z 894.86,A -85,B 0,C 180,E1 -21807.396,E2 -21807.396} C_VEL
LIN {X 0,Y 110.617,Z 904.021,A -85,B 0,C 180,E1 -21812.797,E2 -21812.797} C_VEL
LIN {X 0,Y 97.762,Z 911.622,A -85,B 0,C 180,E1 -21819.912,E2 -21819.912} C_VEL
LIN {X 0,Y 86.579,Z 917.331,A -85,B 0,C 180,E1 -21828.834,E2 -21828.834} C_VEL
LIN {X 0,Y 77.297,Z 921.513,A -85,B 0,C 180,E1 -21840.56,E2 -21840.56} C_VEL
LIN {X 0,Y 71.414,Z 923.944,A -85,B 0,C 180,E1 -21854.575,E2 -21854.575} C_VEL
LIN {X 0,Y 69.408,Z 924.752,A -85,B 0,C 180,E1 -21870.002,E2 -21870.002} C_VEL
LIN {X 0,Y 71.396,Z 923.983,A -85,B 0,C 180,E1 -21885.434,E2 -21885.434} C_VEL
LIN {X 0,Y 77.265,Z 921.586,A -85,B 0,C 180,E1 -21899.458,E2 -21899.458} C_VEL
LIN {X 0,Y 86.535,Z 917.433,A -85,B 0,C 180,E1 -21911.196,E2 -21911.196} C_VEL
LIN {X 0,Y 95.881,Z 912.759,A -85,B 0,C 180,E1 -21918.929,E2 -21918.929} C_VEL
LIN {X 0,Y 77.213,Z 918.425,A -85,B 0,C 180,E1 -21937.138,E2 -21937.138} C_VEL
LIN {X 0,Y 86.051,Z 931.431,A -85,B 0,C 180,E1 -21995.212,E2 -21995.212} C_VEL
LIN {X 0,Y 76.14,Z 937.663,A -85,B 0,C 180,E1 -22005.891,E2 -22005.891} C_VEL
LIN {X 0,Y 69.197,Z 942.645,A -85,B 0,C 180,E1 -22020.572,E2 -22020.572} C_VEL
LIN {X 0,Y 67.18,Z 945.636,A -85,B 0,C 180,E1 -22036.221,E2 -22036.221} C_VEL
LIN {X 0,Y 68.434,Z 946.755,A -85,B 0,C 180,E1 -22048.323,E2 -22048.323} C_VEL
LIN {X 0,Y 68.562,Z 946.797,A -85,B 0,C 180,E1 -22050.833,E2 -22050.833} C_VEL
LIN {X 0,Y 67.078,Z 945.71,A -85,B 0,C 180,E1 -22062.917,E2 -22062.917} C_VEL
LIN {X 0,Y 68.694,Z 942.649,A -85,B 0,C 180,E1 -22079.158,E2 -22079.158} C_VEL
LIN {X 0,Y 74.947,Z 937.754,A -85,B 0,C 180,E1 -22093.923,E2 -22093.923} C_VEL
LIN {X 0,Y 83.613,Z 931.968,A -85,B 0,C 180,E1 -22104.505,E2 -22104.505} C_VEL
LIN {X 0,Y 87.199,Z 929.098,A -85,B 0,C 180,E1 -22108.704,E2 -22108.704} C_VEL
LIN {X 0,Y 95.885,Z 920.528,A -85,B 0,C 180,E1 -22119.609,E2 -22119.609} C_VEL
LIN {X 0,Y 100.035,Z 917.402,A -85,B 0,C 180,E1 -22122.07,E2 -22122.07} C_VEL
LIN {X 0,Y 114.732,Z 906.695,A -85,B 0,C 180,E1 -22127.429,E2 -22127.429} C_VEL
LIN {X 0,Y 129.464,Z 894.378,A -85,B 0,C 180,E1 -22131.315,E2 -22131.315} C_VEL
LIN {X 0,Y 143.712,Z 880.502,A -85,B 0,C 180,E1 -22134.202,E2 -22134.202} C_VEL
LIN {X 0,Y 156.315,Z 866.132,A -85,B 0,C 180,E1 -22136.221,E2 -22136.221} C_VEL
LIN {X 0,Y 168.096,Z 850.244,A -85,B 0,C 180,E1 -22137.812,E2 -22137.812} C_VEL
LIN {X 0,Y 178.55,Z 833.329,A -85,B 0,C 180,E1 -22138.995,E2 -22138.995} C_VEL
LIN {X 0,Y 187.284,Z 816.058,A -85,B 0,C 180,E1 -22139.85,E2 -22139.85} C_VEL
LIN {X 0,Y 193.975,Z 799.616,A -85,B 0,C 180,E1 -22140.426,E2 -22140.426} C_VEL
LIN {X 0,Y 199.371,Z 782.43,A -85,B 0,C 180,E1 -22140.866,E2 -22140.866} C_VEL
LIN {X 0,Y 203.449,Z 763.988,A -85,B 0,C 180,E1 -22141.168,E2 -22141.168} C_VEL
LIN {X 0,Y 208.892,Z 722.093,A -85,B 0,C 180,E1 -22141.874,E2 -22141.874} C_VEL
LIN {X 0,Y 212.765,Z 690.544,A -85,B 0,C 180,E1 -22141.883,E2 -22141.883} C_VEL
LIN {X 0,Y 214.4,Z 677.194,A -85,B 0,C 180,E1 -22141.821,E2 -22141.821} C_VEL
LIN {X 0,Y 217.061,Z 658.474,A -85,B 0,C 180,E1 -22144.426,E2 -22144.426} C_VEL
LIN {X 0,Y 217.289,Z 657.653,A -85,B 0,C 180,E1 -22144.948,E2 -22144.948} C_VEL
LIN {X 0,Y 208.889,Z 728.742,A -85,B 0,C 180,E1 -22146.149,E2 -22146.149} C_VEL
LIN {X 0,Y 204.844,Z 761.467,A -85,B 0,C 180,E1 -22147.082,E2 -22147.082} C_VEL
LIN {X 0,Y 200.746,Z 780.294,A -85,B 0,C 180,E1 -22147.828,E2 -22147.828} C_VEL
LIN {X 0,Y 195.224,Z 797.856,A -85,B 0,C 180,E1 -22148.714,E2 -22148.714} C_VEL
LIN {X 0,Y 188.139,Z 814.891,A -85,B 0,C 180,E1 -22149.792,E2 -22149.792} C_VEL
LIN {X 0,Y 179.826,Z 830.807,A -85,B 0,C 180,E1 -22151.083,E2 -22151.083} C_VEL
LIN {X 0,Y 170.12,Z 846.016,A -85,B 0,C 180,E1 -22152.675,E2 -22152.675} C_VEL
LIN {X 0,Y 159.131,Z 860.315,A -85,B 0,C 180,E1 -22154.625,E2 -22154.625} C_VEL
LIN {X 0,Y 147.399,Z 873.172,A -85,B 0,C 180,E1 -22156.974,E2 -22156.974} C_VEL
LIN {X 0,Y 134.53,Z 885.104,A -85,B 0,C 180,E1 -22159.993,E2 -22159.993} C_VEL
LIN {X 0,Y 120.836,Z 895.839,A -85,B 0,C 180,E1 -22163.921,E2 -22163.921} C_VEL
LIN {X 0,Y 106.529,Z 905.291,A -85,B 0,C 180,E1 -22169.215,E2 -22169.215} C_VEL
LIN {X 0,Y 92.876,Z 912.89,A -85,B 0,C 180,E1 -22176.159,E2 -22176.159} C_VEL
LIN {X 0,Y 80.782,Z 918.598,A -85,B 0,C 180,E1 -22185.133,E2 -22185.133} C_VEL
LIN {X 0,Y 70.508,Z 922.78,A -85,B 0,C 180,E1 -22197.396,E2 -22197.396} C_VEL
LIN {X 0,Y 63.827,Z 925.209,A -85,B 0,C 180,E1 -22212.687,E2 -22212.687} C_VEL
LIN {X 0,Y 61.509,Z 926.015,A -85,B 0,C 180,E1 -22230.003,E2 -22230.003} C_VEL
LIN {X 0,Y 63.808,Z 925.248,A -85,B 0,C 180,E1 -22247.324,E2 -22247.324} C_VEL
LIN {X 0,Y 70.478,Z 922.851,A -85,B 0,C 180,E1 -22262.625,E2 -22262.625} C_VEL
LIN {X 0,Y 80.741,Z 918.698,A -85,B 0,C 180,E1 -22274.902,E2 -22274.902} C_VEL
LIN {X 0,Y 85.318,Z 916.671,A -85,B 0,C 180,E1 -22278.853,E2 -22278.853} C_VEL
LIN {X 0,Y 65.493,Z 923.312,A -85,B 0,C 180,E1 -22305.859,E2 -22305.859} C_VEL
LIN {X 0,Y 76.214,Z 933.139,A -85,B 0,C 180,E1 -22354.916,E2 -22354.916} C_VEL
LIN {X 0,Y 65.879,Z 938.937,A -85,B 0,C 180,E1 -22368.099,E2 -22368.099} C_VEL
LIN {X 0,Y 60.033,Z 943.034,A -85,B 0,C 180,E1 -22385.391,E2 -22385.391} C_VEL
LIN {X 0,Y 59.622,Z 945.128,A -85,B 0,C 180,E1 -22402.287,E2 -22402.287} C_VEL
LIN {X 0,Y 60.705,Z 945.56,A -85,B 0,C 180,E1 -22409.997,E2 -22409.997} C_VEL
LIN {X 0,Y 59.104,Z 944.397,A -85,B 0,C 180,E1 -22424.697,E2 -22424.697} C_VEL
LIN {X 0,Y 61.411,Z 941.414,A -85,B 0,C 180,E1 -22442.496,E2 -22442.496} C_VEL
LIN {X 0,Y 69.135,Z 936.409,A -85,B 0,C 180,E1 -22458.764,E2 -22458.764} C_VEL
LIN {X 0,Y 80.34,Z 929.841,A -85,B 0,C 180,E1 -22470.591,E2 -22470.591} C_VEL
LIN {X 0,Y 94.06,Z 921.378,A -85,B 0,C 180,E1 -22479.295,E2 -22479.295} C_VEL
LIN {X 0,Y 100.035,Z 917.402,A -85,B 0,C 180,E1 -22482.07,E2 -22482.07} C_VEL
LIN {X 0,Y 104.934,Z 913.674,A -85,B 0,C 180,E1 -22484.718,E2 -22484.718} C_VEL
LIN {X 0,Y 115.9,Z 903.606,A -85,B 0,C 180,E1 -22491.746,E2 -22491.746} C_VEL
LIN {X 0,Y 121.15,Z 899.174,A -85,B 0,C 180,E1 -22493.521,E2 -22493.521} C_VEL
LIN {X 0,Y 136.244,Z 885.973,A -85,B 0,C 180,E1 -22496.418,E2 -22496.418} C_VEL
LIN {X 0,Y 150.026,Z 871.728,A -85,B 0,C 180,E1 -22498.53,E2 -22498.53} C_VEL
LIN {X 0,Y 162.185,Z 856.958,A -85,B 0,C 180,E1 -22500.001,E2 -22500.001} C_VEL
LIN {X 0,Y 173.005,Z 841.374,A -85,B 0,C 180,E1 -22501.106,E2 -22501.106} C_VEL
LIN {X 0,Y 182.58,Z 824.749,A -85,B 0,C 180,E1 -22501.975,E2 -22501.975} C_VEL
LIN {X 0,Y 190.669,Z 807.437,A -85,B 0,C 180,E1 -22502.614,E2 -22502.614} C_VEL
LIN {X 0,Y 197.394,Z 788.874,A -85,B 0,C 180,E1 -22503.079,E2 -22503.079} C_VEL
LIN {X 0,Y 202.225,Z 770.537,A -85,B 0,C 180,E1 -22503.371,E2 -22503.371} C_VEL
LIN {X 0,Y 205.525,Z 751.087,A -85,B 0,C 180,E1 -22503.645,E2 -22503.645} C_VEL
LIN {X 0,Y 208.028,Z 731.247,A -85,B 0,C 180,E1 -22504.006,E2 -22504.006} C_VEL
LIN {X 0,Y 203.99,Z 762.825,A -85,B 0,C 180,E1 -22504.88,E2 -22504.88} C_VEL
LIN {X 0,Y 199.823,Z 781.522,A -85,B 0,C 180,E1 -22505.581,E2 -22505.581} C_VEL
LIN {X 0,Y 194.183,Z 799.096,A -85,B 0,C 180,E1 -22506.408,E2 -22506.408} C_VEL
LIN {X 0,Y 187.075,Z 815.9,A -85,B 0,C 180,E1 -22507.389,E2 -22507.389} C_VEL
LIN {X 0,Y 178.499,Z 832.02,A -85,B 0,C 180,E1 -22508.589,E2 -22508.589} C_VEL
LIN {X 0,Y 168.562,Z 847.271,A -85,B 0,C 180,E1 -22510.053,E2 -22510.053} C_VEL
LIN {X 0,Y 157.321,Z 861.573,A -85,B 0,C 180,E1 -22511.838,E2 -22511.838} C_VEL
LIN {X 0,Y 145.287,Z 874.433,A -85,B 0,C 180,E1 -22513.989,E2 -22513.989} C_VEL
LIN {X 0,Y 132.435,Z 886.042,A -85,B 0,C 180,E1 -22516.673,E2 -22516.673} C_VEL
LIN {X 0,Y 118.248,Z 896.829,A -85,B 0,C 180,E1 -22520.286,E2 -22520.286} C_VEL
LIN {X 0,Y 103.277,Z 906.335,A -85,B 0,C 180,E1 -22525.214,E2 -22525.214} C_VEL
LIN {X 0,Y 89.202,Z 913.779,A -85,B 0,C 180,E1 -22531.587,E2 -22531.587} C_VEL
LIN {X 0,Y 76.051,Z 919.584,A -85,B 0,C 180,E1 -22540.315,E2 -22540.315} C_VEL
LIN {X 0,Y 64.497,Z 923.858,A -85,B 0,C 180,E1 -22552.803,E2 -22552.803} C_VEL
LIN {X 0,Y 56.611,Z 926.371,A -85,B 0,C 180,E1 -22569.317,E2 -22569.317} C_VEL
LIN {X 0,Y 53.638,Z 927.238,A -85,B 0,C 180,E1 -22587.866,E2 -22587.866} C_VEL
LIN {X 0,Y 55.524,Z 926.703,A -85,B 0,C 180,E1 -22606.749,E2 -22606.749} C_VEL
LIN {X 0,Y 62.455,Z 924.587,A -85,B 0,C 180,E1 -22624.081,E2 -22624.081} C_VEL
LIN {X 0,Y 73.346,Z 920.747,A -85,B 0,C 180,E1 -22637.406,E2 -22637.406} C_VEL
LIN {X 0,Y 74.862,Z 920.154,A -85,B 0,C 180,E1 -22638.841,E2 -22638.841} C_VEL
LIN {X 0,Y 66.537,Z 934.404,A -85,B 0,C 180,E1 -22714.256,E2 -22714.256} C_VEL
LIN {X 0,Y 56.154,Z 939.583,A -85,B 0,C 180,E1 -22730.129,E2 -22730.129} C_VEL
LIN {X 0,Y 51.465,Z 942.902,A -85,B 0,C 180,E1 -22750.711,E2 -22750.711} C_VEL
LIN {X 0,Y 52.519,Z 944.236,A -85,B 0,C 180,E1 -22768.906,E2 -22768.906} C_VEL
LIN {X 0,Y 52.311,Z 944.17,A -85,B 0,C 180,E1 -22772.188,E2 -22772.188} C_VEL
LIN {X 0,Y 51.331,Z 942.708,A -85,B 0,C 180,E1 -22790.786,E2 -22790.786} C_VEL
LIN {X 0,Y 56.071,Z 939.224,A -85,B 0,C 180,E1 -22811.28,E2 -22811.28} C_VEL
LIN {X 0,Y 66.45,Z 933.783,A -85,B 0,C 180,E1 -22827.413,E2 -22827.413} C_VEL
LIN {X 0,Y 79.696,Z 926.794,A -85,B 0,C 180,E1 -22838.18,E2 -22838.18} C_VEL
LIN {X 0,Y 94.923,Z 917.858,A -85,B 0,C 180,E1 -22845.707,E2 -22845.707} C_VEL
LIN {X 0,Y 110.386,Z 907.403,A -85,B 0,C 180,E1 -22850.851,E2 -22850.851} C_VEL
LIN {X 0,Y 121.15,Z 899.174,A -85,B 0,C 180,E1 -22853.521,E2 -22853.521} C_VEL
LIN {X 0,Y 126.453,Z 894.663,A -85,B 0,C 180,E1 -22855.123,E2 -22855.123} C_VEL
LIN {X 0,Y 138.362,Z 882.664,A -85,B 0,C 180,E1 -22859.869,E2 -22859.869} C_VEL
LIN {X 0,Y 143.407,Z 877.402,A -85,B 0,C 180,E1 -22860.953,E2 -22860.953} C_VEL
LIN {X 0,Y 156.608,Z 862.864,A -85,B 0,C 180,E1 -22862.363,E2 -22862.363} C_VEL
LIN {X 0,Y 168.279,Z 847.615,A -85,B 0,C 180,E1 -22863.453,E2 -22863.453} C_VEL
LIN {X 0,Y 178.97,Z 830.809,A -85,B 0,C 180,E1 -22864.276,E2 -22864.276} C_VEL
LIN {X 0,Y 187.378,Z 814.766,A -85,B 0,C 180,E1 -22864.838,E2 -22864.838} C_VEL
LIN {X 0,Y 178.434,Z 831.745,A -85,B 0,C 180,E1 -22865.951,E2 -22865.951} C_VEL
LIN {X 0,Y 168.324,Z 847.244,A -85,B 0,C 180,E1 -22867.263,E2 -22867.263} C_VEL
LIN {X 0,Y 156.845,Z 861.768,A -85,B 0,C 180,E1 -22868.855,E2 -22868.855} C_VEL
LIN {X 0,Y 144.523,Z 874.809,A -85,B 0,C 180,E1 -22870.77,E2 -22870.77} C_VEL
LIN {X 0,Y 130.791,Z 886.984,A -85,B 0,C 180,E1 -22873.26,E2 -22873.26} C_VEL
LIN {X 0,Y 116.149,Z 897.823,A -85,B 0,C 180,E1 -22876.505,E2 -22876.505} C_VEL
LIN {X 0,Y 101.514,Z 906.851,A -85,B 0,C 180,E1 -22880.662,E2 -22880.662} C_VEL
LIN {X 0,Y 86.144,Z 914.668,A -85,B 0,C 180,E1 -22886.658,E2 -22886.658} C_VEL
LIN {X 0,Y 71.181,Z 920.852,A -85,B 0,C 180,E1 -22895.445,E2 -22895.445} C_VEL
LIN {X 0,Y 58.385,Z 925.124,A -85,B 0,C 180,E1 -22908.1,E2 -22908.1} C_VEL
LIN {X 0,Y 49.291,Z 927.637,A -85,B 0,C 180,E1 -22926.069,E2 -22926.069} C_VEL
LIN {X 0,Y 45.744,Z 928.501,A -85,B 0,C 180,E1 -22947.498,E2 -22947.498} C_VEL
LIN {X 0,Y 48.008,Z 927.967,A -85,B 0,C 180,E1 -22969.469,E2 -22969.469} C_VEL
LIN {X 0,Y 56.073,Z 925.852,A -85,B 0,C 180,E1 -22988.62,E2 -22988.62} C_VEL
